KUKA KRL program: MyProgram_282().src

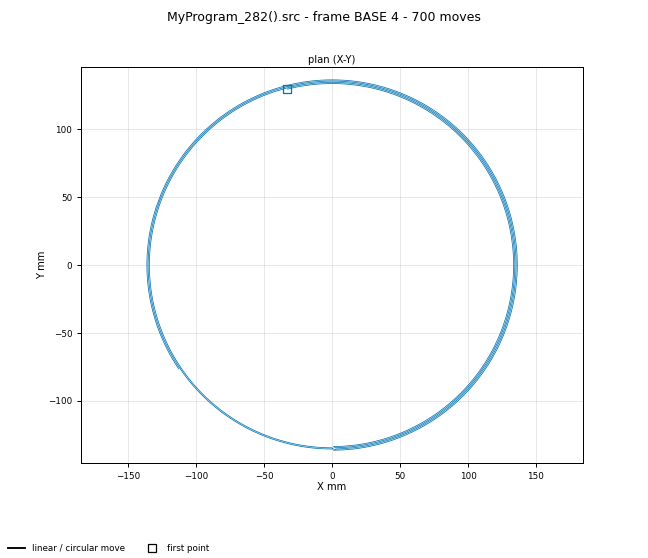
[picture p0: tool path of MyProgram_282().src in frame BASE 4, 700 of 700 moves have a stored position in this frame; points joined in program order, loops and branches not executed]
&ACCESS RVP
&REL 1
&PARAM TEMPLATE = C:\KRC\Roboter\Template\vorgabe
&PARAM EDITMASK = *
DEF MyProgram_282()
; ---- Setting reference (Base) ----
$BASE = BASE_DATA[4]

; --------------------------
; ---- Setting tool (TCP) ----
$TOOL = TOOL_DATA[3]
; --------------------------

$VEL.CP = VEL_APROX_PRINT
Startdeposition()
$VEL.CP = VEL_PRINT
LIN {X -32.8605,Y 129.4603,Z 174,A 104.6033,B 7.9033,C 0.0922,E1 7.8666,E2 347.1729} C_DIS
LIN {X -29.8546,Y 130.1864,Z 174,A 103.1963,B 7.9033,C 0.0926,E1 7.8705,E2 348.5885} C_DIS
LIN {X -26.1954,Y 130.9725,Z 174,A 101.6197,B 7.9033,C 0.0912,E1 7.8748,E2 350.1607} C_DIS
LIN {X -22.189,Y 131.7099,Z 174,A 99.8395,B 7.9033,C 0.0908,E1 7.8797,E2 351.9438} C_DIS
LIN {X -18.2739,Y 132.3113,Z 174,A 98.1779,B 7.9033,C 0.0895,E1 7.8843,E2 353.6} C_DIS
LIN {X -15.2811,Y 132.6899,Z 174,A 96.9189,B 7.9033,C 0.0885,E1 7.8877,E2 354.8542} C_DIS
LIN {X -12.4791,Y 132.9819,Z 174,A 95.5561,B 7.9033,C 0.0906,E1 7.8916,E2 356.2345} C_DIS
LIN {X -8.672,Y 133.2849,Z 174,A 93.9612,B 7.9033,C 0.0896,E1 7.896,E2 357.8234} C_DIS
LIN {X -4.9766,Y 133.4734,Z 174,A 92.4821,B 7.9034,C 0.0876,E1 7.9001,E2 359.289} C_DIS
LIN {X -1.8357,Y 133.5539,Z 174,A 90.9432,B 7.9034,C 0.0906,E1 7.9044,E2 360.8497} C_DIS
LIN {X 2.7143,Y 133.5393,Z 174,A 89.1223,B 7.9034,C 0.0885,E1 7.9095,E2 362.6544} C_DIS
LIN {X 5.81,Y 133.4409,Z 174,A 87.8332,B 7.9034,C 0.088,E1 7.9131,E2 363.9384} C_DIS
LIN {X 8.6689,Y 133.2851,Z 174,A 86.4498,B 7.9034,C 0.0908,E1 7.917,E2 365.3395} C_DIS
LIN {X 12.7986,Y 132.9513,Z 174,A 84.7484,B 7.9034,C 0.09,E1 7.9217,E2 367.0313} C_DIS
LIN {X 17.0686,Y 132.471,Z 174,A 82.9134,B 7.9034,C 0.0904,E1 7.9268,E2 368.8647} C_DIS
LIN {X 20.8861,Y 131.9234,Z 174,A 81.3133,B 7.9034,C 0.0902,E1 7.9312,E2 370.4579} C_DIS
LIN {X 23.9959,Y 131.3934,Z 174,A 79.9828,B 7.9034,C 0.0905,E1 7.9348,E2 371.7853} C_DIS
LIN {X 26.722,Y 130.8653,Z 174,A 78.7856,B 7.9034,C 0.0913,E1 7.9381,E2 372.9829} C_DIS
LIN {X 30.0115,Y 130.1506,Z 174,A 77.2899,B 7.9034,C 0.0931,E1 7.9422,E2 374.4842} C_DIS
LIN {X 35.919,Y 128.6452,Z 174,A 74.2087,B 7.9032,C 0.1029,E1 7.9507,E2 377.6197} C_DIS
LIN {X 40.1681,Y 127.3834,Z 174,A 72.9052,B 7.9033,C 0.0943,E1 7.954,E2 378.8525} C_DIS
LIN {X 44.4232,Y 125.9636,Z 174,A 70.9319,B 7.9033,C 0.0969,E1 7.9592,E2 380.8314} C_DIS
LIN {X 46.9395,Y 125.0457,Z 174,A 69.7782,B 7.9033,C 0.0981,E1 7.9622,E2 381.9855} C_DIS
LIN {X 49.9341,Y 123.8803,Z 174,A 68.3607,B 7.9033,C 0.1002,E1 7.9659,E2 383.4074} C_DIS
LIN {X 53.8065,Y 122.2507,Z 174,A 66.6357,B 7.9033,C 0.1009,E1 7.9703,E2 385.1232} C_DIS
LIN {X 56.4761,Y 121.0388,Z 174,A 65.4067,B 7.9033,C 0.1019,E1 7.9734,E2 386.3488} C_DIS
LIN {X 59.2522,Y 119.7035,Z 174,A 64.0434,B 7.9033,C 0.1043,E1 7.9768,E2 387.7169} C_DIS
LIN {X 62.5045,Y 118.0386,Z 174,A 62.4717,B 7.9032,C 0.1065,E1 7.9807,E2 389.2892} C_DIS
LIN {X 66.3312,Y 115.933,Z 174,A 60.5453,B 7.9032,C 0.11,E1 7.9854,E2 391.222} C_DIS
LIN {X 70.0988,Y 113.6948,Z 174,A 58.7645,B 7.9032,C 0.111,E1 7.9897,E2 392.9911} C_DIS
LIN {X 73.636,Y 111.4363,Z 174,A 56.1409,B 7.9028,C 0.1287,E1 7.996,E2 395.712} C_DIS
LIN {X 78.7721,Y 107.8673,Z 174,A 54.0455,B 7.9029,C 0.1226,E1 8.0006,E2 397.7386} C_DIS
LIN {X 81.3969,Y 105.9004,Z 174,A 53.1152,B 7.903,C 0.1163,E1 8.0026,E2 398.6125} C_DIS
LIN {X 83.7862,Y 104.0199,Z 174,A 51.5738,B 7.903,C 0.123,E1 8.006,E2 400.1825} C_DIS
LIN {X 87.2072,Y 101.1689,Z 174,A 49.5214,B 7.9028,C 0.1291,E1 8.0104,E2 402.2521} C_DIS
LIN {X 90.7533,Y 98.0011,Z 174,A 47.6396,B 7.9028,C 0.1301,E1 8.0142,E2 404.1157} C_DIS
LIN {X 94.316,Y 94.5769,Z 174,A 45.4109,B 7.9028,C 0.1364,E1 8.0187,E2 406.3579} C_DIS
LIN {X 97.4887,Y 91.3036,Z 174,A 43.6195,B 7.9027,C 0.1374,E1 8.0221,E2 408.1304} C_DIS
LIN {X 100.3861,Y 88.108,Z 174,A 41.8763,B 7.9027,C 0.1393,E1 8.0253,E2 409.8615} C_DIS
LIN {X 106.7845,Y 80.2334,Z 174,A 37.8971,B 7.9027,C 0.142,E1 8.0323,E2 413.7978} C_DIS
LIN {X 108.9866,Y 77.2156,Z 174,A 35.9263,B 7.9024,C 0.1527,E1 8.0355,E2 415.8136} C_DIS
LIN {X 111.5979,Y 73.3905,Z 174,A 34.0069,B 7.9024,C 0.1562,E1 8.0385,E2 417.7258} C_DIS
LIN {X 114.0459,Y 69.5264,Z 174,A 32.0466,B 7.9023,C 0.1609,E1 8.0414,E2 419.6868} C_DIS
LIN {X 116.2525,Y 65.7705,Z 174,A 30.1922,B 7.9022,C 0.1653,E1 8.044,E2 421.5405} C_DIS
LIN {X 118.3577,Y 61.8967,Z 174,A 28.4516,B 7.9022,C 0.1672,E1 8.0463,E2 423.264} C_DIS
LIN {X 119.9914,Y 58.6685,Z 174,A 26.8129,B 7.902,C 0.1728,E1 8.0483,E2 424.9141} C_DIS
LIN {X 121.9054,Y 54.5784,Z 174,A 24.9705,B 7.902,C 0.176,E1 8.0504,E2 426.7462} C_DIS
LIN {X 123.4751,Y 50.9311,Z 174,A 23.3908,B 7.9019,C 0.1781,E1 8.0521,E2 428.3122} C_DIS
LIN {X 125.7182,Y 45.1079,Z 174,A 20.7446,B 7.9017,C 0.1847,E1 8.0548,E2 430.9564} C_DIS
LIN {X 126.8147,Y 41.9269,Z 174,A 18.9766,B 7.9015,C 0.195,E1 8.0564,E2 432.7645} C_DIS
LIN {X 127.8659,Y 38.6048,Z 174,A 17.7011,B 7.9015,C 0.1948,E1 8.0574,E2 434.0147} C_DIS
LIN {X 129.0774,Y 34.3337,Z 174,A 15.9304,B 7.9015,C 0.1975,E1 8.0587,E2 435.7705} C_DIS
LIN {X 129.9152,Y 31.0146,Z 174,A 14.4948,B 7.9013,C 0.2009,E1 8.0596,E2 437.2033} C_DIS
LIN {X 130.6576,Y 27.7239,Z 174,A 13.0437,B 7.9013,C 0.2051,E1 8.0605,E2 438.656} C_DIS
LIN {X 131.4588,Y 23.6307,Z 174,A 11.3378,B 7.9012,C 0.2085,E1 8.0614,E2 440.3532} C_DIS
LIN {X 132.0148,Y 20.2961,Z 174,A 9.9295,B 7.9011,C 0.2118,E1 8.062,E2 441.7575} C_DIS
LIN {X 132.5279,Y 16.6348,Z 174,A 8.3933,B 7.901,C 0.2153,E1 8.0626,E2 443.289} C_DIS
LIN {X 132.8256,Y 14.0447,Z 174,A 7.3262,B 7.901,C 0.2175,E1 8.0629,E2 444.3508} C_DIS
LIN {X 133.1108,Y 11.0187,Z 174,A 5.9679,B 7.9008,C 0.2223,E1 8.0632,E2 445.7168} C_DIS
LIN {X 133.38,Y 7.0542,Z 174,A 4.2115,B 7.9006,C 0.2283,E1 8.0635,E2 447.4809} C_DIS
LIN {X 133.5214,Y 3.4601,Z 174,A 2.6915,B 7.9005,C 0.2323,E1 8.0637,E2 448.9995} C_DIS
LIN {X 133.5639,Y -0.9026,Z 174,A 0.8942,B 7.9004,C 0.2362,E1 8.0637,E2 450.7894} C_DIS
LIN {X 133.4787,Y -4.8404,Z 174,A -0.7444,B 7.9003,C 0.2401,E1 8.0635,E2 452.4233} C_DIS
LIN {X 133.2455,Y -9.2583,Z 174,A -2.493,B 7.9002,C 0.2426,E1 8.0633,E2 454.1554} C_DIS
LIN {X 132.9721,Y -12.5819,Z 174,A -3.989,B 7.9,C 0.248,E1 8.0629,E2 455.6608} C_DIS
LIN {X 132.5353,Y -16.5773,Z 174,A -5.793,B 7.8998,C 0.2546,E1 8.0623,E2 457.4761} C_DIS
LIN {X 131.9446,Y -20.7496,Z 174,A -7.4738,B 7.8998,C 0.2572,E1 8.0616,E2 459.1431} C_DIS
LIN {X 131.1931,Y -25.0635,Z 174,A -9.2795,B 7.8996,C 0.2611,E1 8.0607,E2 460.9417} C_DIS
LIN {X 130.4706,Y -28.5898,Z 174,A -11.2579,B 7.8992,C 0.2741,E1 8.0595,E2 462.9744} C_DIS
LIN {X 129.5241,Y -32.609,Z 174,A -13.4588,B 7.8987,C 0.2875,E1 8.058,E2 465.229} C_DIS
LIN {X 127.7535,Y -38.9721,Z 174,A -15.0461,B 7.8993,C 0.2709,E1 8.0569,E2 466.6675} C_DIS
LIN {X 126.3542,Y -43.2965,Z 174,A -17.0965,B 7.899,C 0.2783,E1 8.0551,E2 468.7323} C_DIS
LIN {X 125.4037,Y -45.9802,Z 174,A -18.4062,B 7.8988,C 0.2834,E1 8.0538,E2 470.0541} C_DIS
LIN {X 124.4327,Y -48.5413,Z 174,A -19.6423,B 7.8987,C 0.2878,E1 8.0525,E2 471.2987} C_DIS
LIN {X 122.7297,Y -52.6996,Z 174,A -22.5427,B 7.8978,C 0.312,E1 8.0492,E2 474.3193} C_DIS
LIN {X 119.6529,Y -59.3548,Z 174,A -24.6316,B 7.8982,C 0.2997,E1 8.0468,E2 476.2829} C_DIS
LIN {X 117.5355,Y -63.4486,Z 174,A -27.0607,B 7.8977,C 0.3137,E1 8.0436,E2 478.7694} C_DIS
LIN {X 115.2948,Y -67.4346,Z 174,A -28.5676,B 7.8978,C 0.3098,E1 8.0415,E2 480.2227} C_DIS
LIN {X 113.2822,Y -70.7634,Z 174,A -30.2002,B 7.8978,C 0.3133,E1 8.0391,E2 481.8526} C_DIS
LIN {X 111.0915,Y -74.1547,Z 174,A -32.0728,B 7.8974,C 0.3203,E1 8.0362,E2 483.7441} C_DIS
LIN {X 108.8221,Y -77.4473,Z 174,A -33.5927,B 7.8974,C 0.3207,E1 8.0338,E2 485.2418} C_DIS
LIN {X 105.9642,Y -81.3135,Z 174,A -35.6174,B 7.8973,C 0.3248,E1 8.0304,E2 487.2639} C_DIS
LIN {X 103.3829,Y -84.5709,Z 174,A -37.7765,B 7.8968,C 0.3362,E1 8.0266,E2 489.4709} C_DIS
LIN {X 100.559,Y -87.9099,Z 174,A -39.1592,B 7.897,C 0.3309,E1 8.0241,E2 490.7949} C_DIS
LIN {X 97.7749,Y -90.9962,Z 174,A -40.9704,B 7.8968,C 0.3354,E1 8.0207,E2 492.6113} C_DIS
LIN {X 94.5935,Y -94.2993,Z 174,A -43.2946,B 7.8963,C 0.3464,E1 8.0161,E2 494.9812} C_DIS
LIN {X 91.5907,Y -97.218,Z 174,A -44.4878,B 7.8967,C 0.3386,E1 8.0138,E2 496.1019} C_DIS
LIN {X 89.06,Y -99.5418,Z 174,A -46.1353,B 7.8964,C 0.3449,E1 8.0103,E2 497.7723} C_DIS
LIN {X 85.8583,Y -102.3162,Z 174,A -47.9147,B 7.8963,C 0.3477,E1 8.0066,E2 499.5487} C_DIS
LIN {X 80.6674,Y -106.457,Z 174,A -50.7613,B 7.896,C 0.353,E1 8.0003,E2 502.3976} C_DIS
LIN {X 76.336,Y -109.6042,Z 174,A -53.0261,B 7.8959,C 0.3564,E1 7.9952,E2 504.6606} C_DIS
LIN {X 72.5931,Y -112.1183,Z 174,A -54.9381,B 7.8958,C 0.3593,E1 7.9907,E2 506.5715} C_DIS
LIN {X 67.02,Y -115.5361,Z 174,A -58.2995,B 7.8951,C 0.374,E1 7.9825,E2 510.0037} C_DIS
LIN {X 62.4489,Y -118.0678,Z 174,A -59.6683,B 7.8957,C 0.3612,E1 7.9794,E2 511.2669} C_DIS
LIN {X 58.5733,Y -120.0384,Z 174,A -61.6545,B 7.8955,C 0.3661,E1 7.9744,E2 513.2697} C_DIS
LIN {X 55.9982,Y -121.2598,Z 174,A -62.9844,B 7.8953,C 0.3696,E1 7.971,E2 514.6139} C_DIS
LIN {X 52.5607,Y -122.7898,Z 174,A -64.4615,B 7.8953,C 0.3692,E1 7.9672,E2 516.0753} C_DIS
LIN {X 49.6424,Y -123.9978,Z 174,A -65.8929,B 7.8952,C 0.3722,E1 7.9635,E2 517.5172} C_DIS
LIN {X 46.351,Y -125.2662,Z 174,A -67.3152,B 7.8952,C 0.3722,E1 7.9598,E2 518.9295} C_DIS
LIN {X 42.9664,Y -126.4684,Z 174,A -68.8545,B 7.8951,C 0.3739,E1 7.9558,E2 520.4698} C_DIS
LIN {X 40.2953,Y -127.3428,Z 174,A -70.1004,B 7.8951,C 0.3758,E1 7.9524,E2 521.7215} C_DIS
LIN {X 36.0701,Y -128.603,Z 174,A -72.0478,B 7.8949,C 0.3785,E1 7.9472,E2 523.6771} C_DIS
LIN {X 32.3796,Y -129.5823,Z 174,A -73.5717,B 7.8949,C 0.3779,E1 7.9431,E2 525.1881} C_DIS
LIN {X 29.4655,Y -130.2753,Z 174,A -74.7848,B 7.8949,C 0.3776,E1 7.9398,E2 526.393} C_DIS
LIN {X 26.6085,Y -130.8884,Z 174,A -76.0796,B 7.8949,C 0.3792,E1 7.9363,E2 527.6938} C_DIS
LIN {X 23.365,Y -131.5063,Z 174,A -77.5523,B 7.8947,C 0.3811,E1 7.9322,E2 529.1744} C_DIS
LIN {X 19.6691,Y -132.1119,Z 174,A -79.2862,B 7.8946,C 0.3842,E1 7.9274,E2 530.9251} C_DIS
LIN {X 16.1177,Y -132.5901,Z 174,A -80.7356,B 7.8946,C 0.3835,E1 7.9234,E2 532.3645} C_DIS
LIN {X 11.8861,Y -133.0375,Z 174,A -82.3975,B 7.8947,C 0.3814,E1 7.9188,E2 534.0072} C_DIS
LIN {X 9.1903,Y -133.2504,Z 174,A -83.8262,B 7.8945,C 0.3864,E1 7.9147,E2 535.4697} C_DIS
LIN {X 5.1786,Y -133.4655,Z 174,A -85.4054,B 7.8945,C 0.3843,E1 7.9104,E2 537.032} C_DIS
LIN {X 0.9674,Y -133.5612,Z 174,A -86.8361,B 7.8949,C 0.3782,E1 7.9065,E2 538.4169} C_DIS
Enddeposition()
LIN {X 0.9674,Y -133.5612,Z 174,A -86.8361,B 7.8949,C 0.3782,E1 7.9065,E2 538.4169} C_DIS
Startdeposition()
$VEL.CP = VEL_PRINT
LIN {X 2.3813,Y -134.4521,Z 174,A -85.842,B 7.8949,C 0.3759,E1 7.9092,E2 537.4069} C_DIS
LIN {X 8.4172,Y -134.2094,Z 174,A -83.691,B 7.8946,C 0.3827,E1 7.9151,E2 535.3077} C_DIS
LIN {X 14.1408,Y -133.7276,Z 174,A -80.8337,B 7.8949,C 0.3746,E1 7.9232,E2 532.3976} C_DIS
LIN {X 17.6758,Y -133.3063,Z 174,A -79.3415,B 7.8949,C 0.3743,E1 7.9273,E2 530.9077} C_DIS
LIN {X 21.007,Y -132.8226,Z 174,A -77.9448,B 7.8949,C 0.3741,E1 7.9311,E2 529.5149} C_DIS
LIN {X 23.717,Y -132.3649,Z 174,A -76.7694,B 7.895,C 0.3733,E1 7.9344,E2 528.3381} C_DIS
LIN {X 26.9602,Y -131.7426,Z 174,A -75.349,B 7.895,C 0.3721,E1 7.9383,E2 526.9152} C_DIS
LIN {X 30.122,Y -131.0558,Z 174,A -74.0054,B 7.895,C 0.3717,E1 7.9419,E2 525.5751} C_DIS
LIN {X 33.8293,Y -130.1503,Z 174,A -72.2161,B 7.8953,C 0.3674,E1 7.9468,E2 523.7641} C_DIS
LIN {X 37.6768,Y -129.0867,Z 174,A -70.661,B 7.8953,C 0.3686,E1 7.951,E2 522.2262} C_DIS
LIN {X 41.2611,Y -127.9865,Z 174,A -69.0904,B 7.8953,C 0.3675,E1 7.9551,E2 520.6579} C_DIS
LIN {X 44.3458,Y -126.9506,Z 174,A -67.7307,B 7.8953,C 0.3665,E1 7.9587,E2 519.3005} C_DIS
LIN {X 47.4826,Y -125.8109,Z 174,A -66.3275,B 7.8953,C 0.3653,E1 7.9624,E2 517.8986} C_DIS
LIN {X 50.4496,Y -124.6505,Z 174,A -64.9177,B 7.8955,C 0.3627,E1 7.9661,E2 516.4812} C_DIS
LIN {X 53.3913,Y -123.4189,Z 174,A -63.5797,B 7.8955,C 0.3614,E1 7.9695,E2 515.1447} C_DIS
LIN {X 57.2513,Y -121.679,Z 174,A -61.6065,B 7.8958,C 0.3559,E1 7.9746,E2 513.1488} C_DIS
LIN {X 60.8457,Y -119.9195,Z 174,A -60.1362,B 7.8958,C 0.3579,E1 7.9782,E2 511.7067} C_DIS
LIN {X 64.7447,Y -117.8619,Z 174,A -57.9241,B 7.8961,C 0.3488,E1 7.9837,E2 509.4509} C_DIS
LIN {X 67.8779,Y -116.0865,Z 174,A -56.5245,B 7.8961,C 0.349,E1 7.9871,E2 508.0671} C_DIS
LIN {X 71.2194,Y -114.0668,Z 174,A -55.0969,B 7.8961,C 0.3508,E1 7.9904,E2 506.6679} C_DIS
LIN {X 74.4195,Y -112.0055,Z 174,A -53.4031,B 7.8962,C 0.3468,E1 7.9944,E2 504.9635} C_DIS
LIN {X 78.1874,Y -109.4081,Z 174,A -51.4969,B 7.8963,C 0.3442,E1 7.9987,E2 503.0612} C_DIS
LIN {X 82.2337,Y -106.4004,Z 174,A -49.2415,B 7.8966,C 0.3382,E1 8.0038,E2 500.7903} C_DIS
LIN {X 85.1332,Y -104.0948,Z 174,A -47.7998,B 7.8966,C 0.3378,E1 8.0069,E2 499.3644} C_DIS
LIN {X 88.4233,Y -101.3149,Z 174,A -45.9787,B 7.8967,C 0.3345,E1 8.0107,E2 497.5434} C_DIS
LIN {X 91.8873,Y -98.1847,Z 174,A -43.8328,B 7.897,C 0.3274,E1 8.0152,E2 495.3758} C_DIS
LIN {X 95.0883,Y -95.0883,Z 174,A -42.2035,B 7.897,C 0.3287,E1 8.0183,E2 493.7786} C_DIS
LIN {X 97.9798,Y -92.1054,Z 174,A -40.4175,B 7.8972,C 0.3245,E1 8.0218,E2 491.9888} C_DIS
LIN {X 100.9496,Y -88.8407,Z 174,A -38.3676,B 7.8975,C 0.317,E1 8.0256,E2 489.9158} C_DIS
LIN {X 103.8494,Y -85.4336,Z 174,A -36.7918,B 7.8974,C 0.3192,E1 8.0284,E2 488.3798} C_DIS
LIN {X 106.1126,Y -82.6051,Z 174,A -34.9879,B 7.8977,C 0.3104,E1 8.0316,E2 486.5415} C_DIS
LIN {X 108.9982,Y -78.758,Z 174,A -32.7842,B 7.898,C 0.3025,E1 8.0352,E2 484.3163} C_DIS
LIN {X 111.3244,Y -75.4339,Z 174,A -31.7902,B 7.8976,C 0.3129,E1 8.0367,E2 483.413} C_DIS
LIN {X 112.9455,Y -72.9849,Z 174,A -30.1105,B 7.8981,C 0.3013,E1 8.0393,E2 481.6784} C_DIS
LIN {X 114.9785,Y -69.738,Z 174,A -28.6361,B 7.8981,C 0.3003,E1 8.0414,E2 480.2222} C_DIS
LIN {X 118.6158,Y -63.3546,Z 174,A -25.506,B 7.8984,C 0.2923,E1 8.0457,E2 477.0891} C_DIS
LIN {X 121.6414,Y -57.3288,Z 174,A -22.2905,B 7.8989,C 0.2779,E1 8.0497,E2 473.8275} C_DIS
LIN {X 123.3919,Y -53.4539,Z 174,A -21.2791,B 7.8985,C 0.2891,E1 8.0507,E2 472.9147} C_DIS
LIN {X 124.8493,Y -49.9564,Z 174,A -19.4436,B 7.8988,C 0.2803,E1 8.0527,E2 471.0501} C_DIS
LIN {X 125.9847,Y -47.0186,Z 174,A -18.1067,B 7.899,C 0.2767,E1 8.054,E2 469.7125} C_DIS
LIN {X 127.049,Y -44.0619,Z 174,A -16.7581,B 7.899,C 0.2729,E1 8.0553,E2 468.3614} C_DIS
LIN {X 128.2227,Y -40.5219,Z 174,A -15.1119,B 7.8993,C 0.2673,E1 8.0567,E2 466.7065} C_DIS
LIN {X 130.3883,Y -32.8914,Z 174,A -11.9004,B 7.8995,C 0.2612,E1 8.0591,E2 463.5128} C_DIS
LIN {X 131.0796,Y -30.0178,Z 174,A -10.6649,B 7.8995,C 0.2582,E1 8.0598,E2 462.2791} C_DIS
LIN {X 131.7739,Y -26.8062,Z 174,A -9.2631,B 7.8997,C 0.2541,E1 8.0606,E2 460.8758} C_DIS
LIN {X 132.4425,Y -23.2829,Z 174,A -7.6806,B 7.8999,C 0.2487,E1 8.0614,E2 459.285} C_DIS
LIN {X 133.1232,Y -19.0049,Z 174,A -5.9996,B 7.8999,C 0.2467,E1 8.0621,E2 457.6228} C_DIS
LIN {X 133.5736,Y -15.5317,Z 174,A -4.5641,B 7.9,C 0.2436,E1 8.0626,E2 456.193} C_DIS
LIN {X 133.9202,Y -12.1981,Z 174,A -3.135,B 7.9002,C 0.2394,E1 8.063,E2 454.7624} C_DIS
LIN {X 134.3453,Y -5.8976,Z 174,A -0.5351,B 7.9003,C 0.2335,E1 8.0635,E2 452.1714} C_DIS
LIN {X 134.4584,Y -2.0056,Z 174,A 1.1198,B 7.9005,C 0.2288,E1 8.0635,E2 450.5155} C_DIS
LIN {X 134.4696,Y 1.1061,Z 174,A 2.4735,B 7.9006,C 0.2244,E1 8.0635,E2 449.1573} C_DIS
LIN {X 134.3394,Y 6.036,Z 174,A 4.4801,B 7.9007,C 0.2203,E1 8.0634,E2 447.1606} C_DIS
LIN {X 134.071,Y 10.4088,Z 174,A 6.3941,B 7.9009,C 0.2139,E1 8.063,E2 445.2392} C_DIS
LIN {X 133.7055,Y 14.3466,Z 174,A 8.0408,B 7.901,C 0.2099,E1 8.0626,E2 443.5958} C_DIS
LIN {X 133.2842,Y 17.8447,Z 174,A 9.5869,B 7.9011,C 0.2047,E1 8.062,E2 442.0429} C_DIS
LIN {X 132.6696,Y 21.9493,Z 174,A 11.238,B 7.9012,C 0.202,E1 8.0613,E2 440.4049} C_DIS
LIN {X 132.0391,Y 25.4689,Z 174,A 12.7066,B 7.9012,C 0.1988,E1 8.0605,E2 438.9419} C_DIS
LIN {X 131.3327,Y 28.8953,Z 174,A 14.17,B 7.9014,C 0.1952,E1 8.0597,E2 437.4807} C_DIS
LIN {X 130.4583,Y 32.6158,Z 174,A 15.8511,B 7.9015,C 0.1896,E1 8.0586,E2 435.7919} C_DIS
LIN {X 129.4257,Y 36.4964,Z 174,A 17.4995,B 7.9015,C 0.1861,E1 8.0574,E2 434.15} C_DIS
LIN {X 128.0732,Y 40.9899,Z 174,A 19.4535,B 7.9017,C 0.1815,E1 8.0558,E2 432.2002} C_DIS
LIN {X 126.8433,Y 44.6551,Z 174,A 21.7743,B 7.9021,C 0.1636,E1 8.0536,E2 429.7949} C_DIS
LIN {X 124.8933,Y 49.8474,Z 174,A 23.2295,B 7.9018,C 0.1753,E1 8.0522,E2 428.4506} C_DIS
LIN {X 123.3919,Y 53.4539,Z 174,A 25.0313,B 7.902,C 0.1682,E1 8.0502,E2 426.6308} C_DIS
LIN {X 121.9697,Y 56.6241,Z 174,A 26.4792,B 7.902,C 0.165,E1 8.0485,E2 425.186} C_DIS
LIN {X 120.3103,Y 60.0725,Z 174,A 28.033,B 7.9021,C 0.1623,E1 8.0466,E2 423.6407} C_DIS
LIN {X 119.1138,Y 62.4081,Z 174,A 29.1522,B 7.9021,C 0.1594,E1 8.0452,E2 422.5207} C_DIS
LIN {X 117.0655,Y 66.1754,Z 174,A 31.0938,B 7.9023,C 0.1526,E1 8.0425,E2 420.5641} C_DIS
LIN {X 114.7688,Y 70.0828,Z 174,A 32.9901,B 7.9023,C 0.1486,E1 8.0398,E2 418.6711} C_DIS
LIN {X 112.2911,Y 73.9872,Z 174,A 34.8991,B 7.9025,C 0.145,E1 8.0369,E2 416.7687} C_DIS
LIN {X 109.719,Y 77.7506,Z 174,A 36.7459,B 7.9025,C 0.1423,E1 8.034,E2 414.9326} C_DIS
LIN {X 107.2283,Y 81.1512,Z 174,A 38.9497,B 7.9027,C 0.1303,E1 8.0302,E2 412.678} C_DIS
LIN {X 104.6851,Y 84.4061,Z 174,A 40.4134,B 7.9027,C 0.1321,E1 8.0277,E2 411.2501} C_DIS
LIN {X 102.145,Y 87.4639,Z 174,A 42.0062,B 7.9027,C 0.1303,E1 8.0249,E2 409.669} C_DIS
LIN {X 99.1956,Y 90.7949,Z 174,A 43.8858,B 7.9027,C 0.1266,E1 8.0214,E2 407.7907} C_DIS
LIN {X 95.8545,Y 94.3152,Z 174,A 45.6568,B 7.9027,C 0.128,E1 8.018,E2 406.0553} C_DIS
LIN {X 92.6153,Y 97.4985,Z 174,A 47.8455,B 7.9029,C 0.1193,E1 8.0136,E2 403.8352} C_DIS
LIN {X 89.0835,Y 100.735,Z 174,A 49.7474,B 7.9029,C 0.118,E1 8.0096,E2 401.9497} C_DIS
LIN {X 86.0762,Y 103.3172,Z 174,A 51.4874,B 7.9029,C 0.114,E1 8.0059,E2 400.2031} C_DIS
LIN {X 82.7455,Y 106.0035,Z 174,A 53.3315,B 7.903,C 0.1103,E1 8.0019,E2 398.3562} C_DIS
LIN {X 80.0111,Y 108.0822,Z 174,A 54.7695,B 7.903,C 0.1083,E1 7.9987,E2 396.921} C_DIS
LIN {X 75.6484,Y 111.1792,Z 174,A 57.0117,B 7.903,C 0.1053,E1 7.9935,E2 394.6831} C_DIS
LIN {X 71.9678,Y 113.5962,Z 174,A 58.8795,B 7.9031,C 0.1025,E1 7.9891,E2 392.8161} C_DIS
LIN {X 68.0663,Y 115.9758,Z 174,A 60.7919,B 7.9031,C 0.1003,E1 7.9846,E2 390.9079} C_DIS
LIN {X 64.0541,Y 118.2397,Z 174,A 62.7306,B 7.9031,C 0.098,E1 7.9798,E2 388.9721} C_DIS
LIN {X 60.8995,Y 119.8921,Z 174,A 64.1407,B 7.9031,C 0.098,E1 7.9764,E2 387.5749} C_DIS
LIN {X 58.0887,Y 121.279,Z 174,A 65.5291,B 7.9032,C 0.0953,E1 7.9729,E2 386.1801} C_DIS
LIN {X 54.8131,Y 122.7941,Z 174,A 67.0554,B 7.9032,C 0.0937,E1 7.969,E2 384.6552} C_DIS
LIN {X 51.3445,Y 124.2855,Z 174,A 68.7308,B 7.9032,C 0.0908,E1 7.9647,E2 382.9719} C_DIS
LIN {X 47.7987,Y 125.6926,Z 174,A 70.2135,B 7.9032,C 0.0916,E1 7.9608,E2 381.5067} C_DIS
LIN {X 43.8151,Y 127.1345,Z 174,A 72.0448,B 7.9032,C 0.0894,E1 7.956,E2 379.6725} C_DIS
LIN {X 37.4065,Y 129.1659,Z 174,A 74.869,B 7.9032,C 0.0878,E1 7.9485,E2 376.8537} C_DIS
LIN {X 34.4529,Y 129.9844,Z 174,A 76.1582,B 7.9032,C 0.0871,E1 7.945,E2 375.5668} C_DIS
LIN {X 31.121,Y 130.8227,Z 174,A 77.5904,B 7.9033,C 0.0866,E1 7.9411,E2 374.1388} C_DIS
LIN {X 27.4201,Y 131.649,Z 174,A 79.3043,B 7.9033,C 0.084,E1 7.9364,E2 372.4135} C_DIS
LIN {X 23.7136,Y 132.3655,Z 174,A 80.8085,B 7.9033,C 0.0849,E1 7.9323,E2 370.9223} C_DIS
LIN {X 19.8449,Y 133.0026,Z 174,A 82.625,B 7.9033,C 0.0817,E1 7.9273,E2 369.0888} C_DIS
LIN {X 16.0053,Y 133.5171,Z 174,A 84.1357,B 7.9033,C 0.0835,E1 7.9231,E2 367.5954} C_DIS
LIN {X 12.5603,Y 133.8854,Z 174,A 85.601,B 7.9033,C 0.0832,E1 7.9191,E2 366.1319} C_DIS
LIN {X 8.953,Y 134.1764,Z 174,A 87.2671,B 7.9033,C 0.0809,E1 7.9144,E2 364.4515} C_DIS
LIN {X 4.969,Y 134.3815,Z 174,A 88.8768,B 7.9033,C 0.0822,E1 7.9099,E2 362.8534} C_DIS
LIN {X -0.5309,Y 134.4723,Z 174,A 91.219,B 7.9033,C 0.0822,E1 7.9034,E2 360.5125} C_DIS
LIN {X -4.0382,Y 134.4128,Z 174,A 92.8113,B 7.9033,C 0.0806,E1 7.8989,E2 358.9091} C_DIS
LIN {X -8.3743,Y 134.2121,Z 174,A 94.5206,B 7.9033,C 0.0832,E1 7.8942,E2 357.2175} C_DIS
LIN {X -12.2442,Y 133.9158,Z 174,A 96.3017,B 7.9033,C 0.0816,E1 7.8892,E2 355.4221} C_DIS
LIN {X -16.1828,Y 133.4959,Z 174,A 97.8683,B 7.9033,C 0.0841,E1 7.8849,E2 353.8708} C_DIS
LIN {X -19.1868,Y 133.0972,Z 174,A 99.1997,B 7.9033,C 0.084,E1 7.8812,E2 352.5354} C_DIS
LIN {X -22.3361,Y 132.605,Z 174,A 100.5591,B 7.9033,C 0.0846,E1 7.8775,E2 351.1766} C_DIS
LIN {X -26.3997,Y 131.8566,Z 174,A 102.3847,B 7.9033,C 0.0846,E1 7.8724,E2 349.3442} C_DIS
LIN {X -30.1179,Y 131.0567,Z 174,A 103.9525,B 7.9033,C 0.0864,E1 7.8682,E2 347.7837} C_DIS
LIN {X -33.4639,Y 130.243,Z 174,A 105.4104,B 7.9033,C 0.0876,E1 7.8642,E2 346.328} C_DIS
LIN {X -42.2849,Y 127.6516,Z 174,A 110.6048,B 7.9035,C 0.0708,E1 7.85,E2 340.9811} C_DIS
LIN {X -50.053,Y 124.8104,Z 174,A 112.9823,B 7.9032,C 0.0925,E1 7.8442,E2 338.746} C_DIS
LIN {X -53.7812,Y 123.2504,Z 174,A 114.6321,B 7.9032,C 0.0955,E1 7.84,E2 337.1061} C_DIS
LIN {X -57.5211,Y 121.5501,Z 174,A 117.135,B 7.9033,C 0.0862,E1 7.8334,E2 334.5136} C_DIS
LIN {X -62.4517,Y 119.0909,Z 174,A 118.7522,B 7.9031,C 0.1004,E1 7.8296,E2 332.9867} C_DIS
LIN {X -66.276,Y 117.0088,Z 174,A 120.6779,B 7.9031,C 0.102,E1 7.8249,E2 331.0542} C_DIS
LIN {X -69.7149,Y 114.9924,Z 174,A 122.5742,B 7.9031,C 0.1016,E1 7.8203,E2 329.1354} C_DIS
LIN {X -73.5924,Y 112.551,Z 174,A 124.4486,B 7.9031,C 0.1058,E1 7.8159,E2 327.2721} C_DIS
LIN {X -78.2444,Y 109.3674,Z 174,A 126.8243,B 7.9031,C 0.1102,E1 7.8105,E2 324.9016} C_DIS
LIN {X -81.2312,Y 107.1679,Z 174,A 128.3699,B 7.903,C 0.1134,E1 7.8071,E2 323.3616} C_DIS
LIN {X -84.4073,Y 104.6843,Z 174,A 130.0713,B 7.903,C 0.1168,E1 7.8033,E2 321.6637} C_DIS
LIN {X -87.4332,Y 102.1715,Z 174,A 132.1851,B 7.903,C 0.1135,E1 7.7987,E2 319.4986} C_DIS
LIN {X -90.2359,Y 99.7041,Z 174,A 133.3286,B 7.9028,C 0.1231,E1 7.7965,E2 318.4106} C_DIS
LIN {X -92.9859,Y 97.1443,Z 174,A 135.2172,B 7.9028,C 0.1222,E1 7.7926,E2 316.4888} C_DIS
LIN {X -95.8367,Y 94.3334,Z 174,A 136.8478,B 7.9028,C 0.1268,E1 7.7894,E2 314.8689} C_DIS
LIN {X -99.5704,Y 90.3833,Z 174,A 139.006,B 7.9026,C 0.134,E1 7.7853,E2 312.7319} C_DIS
LIN {X -102.0372,Y 87.5891,Z 174,A 140.8975,B 7.9026,C 0.1331,E1 7.7818,E2 310.8054} C_DIS
LIN {X -104.3536,Y 84.8166,Z 174,A 142.3734,B 7.9026,C 0.1375,E1 7.7792,E2 309.3386} C_DIS
LIN {X -107.1068,Y 81.3123,Z 174,A 144.2931,B 7.9026,C 0.1415,E1 7.7759,E2 307.4182} C_DIS
LIN {X -109.554,Y 77.9834,Z 174,A 146.0587,B 7.9024,C 0.1456,E1 7.773,E2 305.6536} C_DIS
LIN {X -112.0702,Y 74.3225,Z 174,A 147.9557,B 7.9024,C 0.1501,E1 7.7701,E2 303.758} C_DIS
LIN {X -114.6831,Y 70.2222,Z 174,A 150.219,B 7.9024,C 0.1525,E1 7.7667,E2 301.4735} C_DIS
LIN {X -116.9969,Y 66.2967,Z 174,A 152.4472,B 7.9023,C 0.1534,E1 7.7635,E2 299.2123} C_DIS
LIN {X -118.8895,Y 62.8353,Z 174,A 153.5059,B 7.902,C 0.1664,E1 7.7623,E2 298.2308} C_DIS
LIN {X -120.648,Y 59.388,Z 174,A 155.3959,B 7.902,C 0.1673,E1 7.7598,E2 296.3132} C_DIS
LIN {X -122.1317,Y 56.2738,Z 174,A 156.8719,B 7.902,C 0.1711,E1 7.7581,E2 294.838} C_DIS
LIN {X -123.5734,Y 53.0341,Z 174,A 158.4305,B 7.9019,C 0.1744,E1 7.7563,E2 293.275} C_DIS
LIN {X -125.2331,Y 48.986,Z 174,A 160.9132,B 7.9019,C 0.1709,E1 7.7537,E2 290.7188} C_DIS
LIN {X -126.9254,Y 44.4184,Z 174,A 162.2385,B 7.9016,C 0.1869,E1 7.7526,E2 289.4869} C_DIS
LIN {X -128.222,Y 40.524,Z 174,A 164.1958,B 7.9016,C 0.1889,E1 7.7508,E2 287.5061} C_DIS
LIN {X -129.2305,Y 37.1856,Z 174,A 165.6964,B 7.9014,C 0.1928,E1 7.7497,E2 286.0052} C_DIS
LIN {X -130.0577,Y 34.1782,Z 174,A 167.0568,B 7.9014,C 0.1961,E1 7.7487,E2 284.6422} C_DIS
LIN {X -130.7645,Y 31.3625,Z 174,A 168.327,B 7.9013,C 0.1991,E1 7.7478,E2 283.3691} C_DIS
LIN {X -131.657,Y 27.3807,Z 174,A 170.175,B 7.9012,C 0.2025,E1 7.7467,E2 281.5095} C_DIS
LIN {X -132.349,Y 23.8058,Z 174,A 171.6825,B 7.9011,C 0.2075,E1 7.746,E2 280.0088} C_DIS
LIN {X -132.9284,Y 20.3242,Z 174,A 173.2849,B 7.901,C 0.2105,E1 7.7453,E2 278.3958} C_DIS
LIN {X -133.5099,Y 16.0657,Z 174,A 175.0881,B 7.9008,C 0.2161,E1 7.7446,E2 276.5977} C_DIS
LIN {X -133.9018,Y 12.3901,Z 174,A 176.7815,B 7.9008,C 0.219,E1 7.7441,E2 274.8913} C_DIS
LIN {X -134.2173,Y 8.2887,Z 174,A 178.471,B 7.9006,C 0.2249,E1 7.7438,E2 273.2111} C_DIS
LIN {X -134.395,Y 4.6238,Z 174,A -179.8037,B 7.9006,C 0.2272,E1 7.7436,E2 271.4675} C_DIS
LIN {X -134.4765,Y 0.1063,Z 174,A -177.8878,B 7.9004,C 0.2329,E1 7.7436,E2 269.5544} C_DIS
LIN {X -134.4198,Y -3.7854,Z 174,A -176.297,B 7.9002,C 0.2386,E1 7.7436,E2 267.9732} C_DIS
LIN {X -134.2674,Y -7.4689,Z 174,A -174.5566,B 7.9002,C 0.2408,E1 7.7439,E2 266.2134} C_DIS
LIN {X -133.9841,Y -11.4568,Z 174,A -172.9515,B 7.8999,C 0.247,E1 7.7443,E2 264.6217} C_DIS
LIN {X -133.6903,Y -14.4878,Z 174,A -171.5928,B 7.8999,C 0.2499,E1 7.7447,E2 263.2567} C_DIS
LIN {X -133.1721,Y -18.6626,Z 174,A -169.7202,B 7.8997,C 0.2539,E1 7.7454,E2 261.3757} C_DIS
LIN {X -132.5898,Y -22.4271,Z 174,A -168.1743,B 7.8995,C 0.2596,E1 7.746,E2 259.8406} C_DIS
LIN {X -131.9805,Y -25.7756,Z 174,A -166.6562,B 7.8995,C 0.2627,E1 7.7468,E2 258.3152} C_DIS
LIN {X -131.187,Y -29.5476,Z 174,A -164.3928,B 7.8995,C 0.2587,E1 7.7483,E2 255.9763} C_DIS
LIN {X -130.0374,Y -34.2544,Z 174,A -162.859,B 7.8991,C 0.2718,E1 7.7493,E2 254.5097} C_DIS
LIN {X -128.241,Y -40.4645,Z 174,A -160.238,B 7.8988,C 0.2812,E1 7.7514,E2 251.9072} C_DIS
LIN {X -126.9395,Y -44.3777,Z 174,A -158.1978,B 7.8988,C 0.282,E1 7.7532,E2 249.8333} C_DIS
LIN {X -125.7762,Y -47.5753,Z 174,A -156.8476,B 7.8986,C 0.2873,E1 7.7545,E2 248.4964} C_DIS
LIN {X -124.6749,Y -50.389,Z 174,A -155.5745,B 7.8985,C 0.2909,E1 7.7558,E2 247.2258} C_DIS
LIN {X -123.3315,Y -53.5935,Z 174,A -153.9703,B 7.8984,C 0.293,E1 7.7576,E2 245.6073} C_DIS
LIN {X -120.6633,Y -59.357,Z 174,A -151.4685,B 7.898,C 0.3029,E1 7.7605,E2 243.1324} C_DIS
LIN {X -118.9991,Y -62.6265,Z 174,A -148.8803,B 7.8984,C 0.2921,E1 7.7641,E2 240.4177} C_DIS
LIN {X -116.1285,Y -67.8064,Z 174,A -147.2994,B 7.8977,C 0.312,E1 7.7661,E2 238.9556} C_DIS
LIN {X -113.7521,Y -71.7208,Z 174,A -145.0274,B 7.8977,C 0.312,E1 7.7695,E2 236.6449} C_DIS
LIN {X -110.1713,Y -77.1091,Z 174,A -142.2408,B 7.8974,C 0.318,E1 7.7738,E2 233.8559} C_DIS
LIN {X -107.8152,Y -80.3696,Z 174,A -140.1711,B 7.8974,C 0.3167,E1 7.7773,E2 231.7426} C_DIS
LIN {X -105.4426,Y -83.459,Z 174,A -139.0476,B 7.897,C 0.3283,E1 7.7792,E2 230.6866} C_DIS
LIN {X -103.3592,Y -86.0255,Z 174,A -137.3616,B 7.897,C 0.3272,E1 7.7822,E2 228.9666} C_DIS
LIN {X -100.1573,Y -89.7325,Z 174,A -135.4835,B 7.8967,C 0.3347,E1 7.7856,E2 227.1153} C_DIS
LIN {X -97.3539,Y -92.7667,Z 174,A -133.7883,B 7.8965,C 0.3393,E1 7.7888,E2 225.4288} C_DIS
LIN {X -95.1856,Y -94.9904,Z 174,A -132.1045,B 7.8967,C 0.3365,E1 7.7922,E2 223.7005} C_DIS
LIN {X -91.9977,Y -98.0813,Z 174,A -130.2462,B 7.8965,C 0.3406,E1 7.7959,E2 221.8469} C_DIS
LIN {X -89.0056,Y -100.8038,Z 174,A -128.5053,B 7.8964,C 0.3435,E1 7.7996,E2 220.1042} C_DIS
LIN {X -85.6437,Y -103.6753,Z 174,A -126.0884,B 7.8966,C 0.3387,E1 7.8049,E2 217.6209} C_DIS
LIN {X -81.9363,Y -106.6299,Z 174,A -123.8236,B 7.8966,C 0.3383,E1 7.81,E2 215.3256} C_DIS
LIN {X -77.1785,Y -110.1229,Z 174,A -122.0345,B 7.8959,C 0.3535,E1 7.8139,E2 213.6281} C_DIS
LIN {X -73.6159,Y -112.5356,Z 174,A -120.1102,B 7.8959,C 0.3549,E1 7.8184,E2 211.6927} C_DIS
LIN {X -69.8751,Y -114.8955,Z 174,A -118.2017,B 7.8957,C 0.3572,E1 7.8229,E2 209.7812} C_DIS
LIN {X -65.979,Y -117.1759,Z 174,A -116.3039,B 7.8957,C 0.3602,E1 7.8275,E2 207.8867} C_DIS
LIN {X -62.2518,Y -119.1958,Z 174,A -114.572,B 7.8955,C 0.3636,E1 7.8317,E2 206.164} C_DIS
LIN {X -58.9149,Y -120.8813,Z 174,A -112.9803,B 7.8954,C 0.3655,E1 7.8357,E2 204.5725} C_DIS
LIN {X -56.1724,Y -122.1786,Z 174,A -111.6484,B 7.8954,C 0.3663,E1 7.8391,E2 203.2356} C_DIS
LIN {X -52.2686,Y -123.8996,Z 174,A -109.972,B 7.8951,C 0.3705,E1 7.8434,E2 201.5768} C_DIS
LIN {X -49.1087,Y -125.1854,Z 174,A -108.2002,B 7.8953,C 0.3667,E1 7.8481,E2 199.7649} C_DIS
LIN {X -44.7873,Y -126.7975,Z 174,A -105.8339,B 7.8955,C 0.3619,E1 7.8544,E2 197.3477} C_DIS
LIN {X -40.4688,Y -128.2396,Z 174,A -104.3872,B 7.8951,C 0.3715,E1 7.8581,E2 195.963} C_DIS
LIN {X -37.4138,Y -129.1637,Z 174,A -103.1151,B 7.895,C 0.3739,E1 7.8615,E2 194.7016} C_DIS
LIN {X -34.4249,Y -129.9919,Z 174,A -101.7714,B 7.895,C 0.3743,E1 7.8651,E2 193.3548} C_DIS
LIN {X -31.0909,Y -130.8299,Z 174,A -100.2935,B 7.895,C 0.375,E1 7.8691,E2 191.8749} C_DIS
LIN {X -27.4755,Y -131.6377,Z 174,A -98.59,B 7.895,C 0.3737,E1 7.8738,E2 190.1553} C_DIS
LIN {X -23.5254,Y -132.3991,Z 174,A -96.9652,B 7.8949,C 0.3758,E1 7.8782,E2 188.5412} C_DIS
LIN {X -19.5884,Y -133.0398,Z 174,A -95.193,B 7.8949,C 0.3752,E1 7.8832,E2 186.7593} C_DIS
LIN {X -14.5095,Y -133.688,Z 174,A -93.1004,B 7.8949,C 0.3772,E1 7.8889,E2 184.677} C_DIS
LIN {X -11.0853,Y -134.0155,Z 174,A -91.6286,B 7.8949,C 0.3772,E1 7.893,E2 183.2039} C_DIS
LIN {X -7.0776,Y -134.2871,Z 174,A -89.556,B 7.8951,C 0.3711,E1 7.8989,E2 181.085} C_DIS
LIN {X -3.5219,Y -134.4271,Z 174,A -88.0934,B 7.8951,C 0.372,E1 7.903,E2 179.6285} C_DIS
LIN {X -0.1286,Y -134.4745,Z 174,A -87.046,B 7.8948,C 0.3788,E1 7.9058,E2 178.6308} C_DIS
LIN {X -0.1286,Y -134.4745,Z 174,A -87.046,B 7.8948,C 0.3788,E1 7.9058,E2 178.6308} C_DIS
Enddeposition()
LIN {X 0.989,Y -135.3751,Z 174,A -86.4984,B 7.8336,C 0.3827,E1 7.8463,E2 178.1248} C_DIS
Startdeposition()
$VEL.CP = VEL_PRINT
LIN {X -4.5948,Y -135.3035,Z 174,A -89.4877,B 7.8331,C 0.3937,E1 7.8378,E2 181.1943} C_DIS
LIN {X -9.3622,Y -135.0569,Z 174,A -91.5179,B 7.8331,C 0.3937,E1 7.8321,E2 183.2266} C_DIS
LIN {X -13.7953,Y -134.6772,Z 174,A -93.5276,B 7.833,C 0.3956,E1 7.8265,E2 185.2529} C_DIS
LIN {X -18.3201,Y -134.1368,Z 174,A -95.35,B 7.8331,C 0.3934,E1 7.8215,E2 187.0628} C_DIS
LIN {X -22.2045,Y -133.5467,Z 174,A -96.9742,B 7.8331,C 0.3922,E1 7.817,E2 188.6825} C_DIS
LIN {X -26.3145,Y -132.7997,Z 174,A -98.8098,B 7.8331,C 0.3926,E1 7.8119,E2 190.5272} C_DIS
LIN {X -29.9985,Y -132.0145,Z 174,A -100.256,B 7.8333,C 0.3893,E1 7.808,E2 191.9553} C_DIS
LIN {X -33.2623,Y -131.2301,Z 174,A -101.7189,B 7.8333,C 0.3892,E1 7.8041,E2 193.4238} C_DIS
LIN {X -36.4956,Y -130.3679,Z 174,A -103.1531,B 7.8333,C 0.3886,E1 7.8002,E2 194.8606} C_DIS
LIN {X -39.1562,Y -129.5944,Z 174,A -104.9344,B 7.8329,C 0.3976,E1 7.7952,E2 196.718} C_DIS
LIN {X -43.8313,Y -128.089,Z 174,A -106.4895,B 7.8334,C 0.3875,E1 7.7913,E2 198.2084} C_DIS
LIN {X -47.1577,Y -126.9013,Z 174,A -107.7591,B 7.8336,C 0.3826,E1 7.788,E2 199.4499} C_DIS
LIN {X -50.7926,Y -125.4903,Z 174,A -109.5662,B 7.8336,C 0.3835,E1 7.7833,E2 201.2769} C_DIS
LIN {X -53.9418,Y -124.1692,Z 174,A -111.1459,B 7.8336,C 0.3842,E1 7.7792,E2 202.8735} C_DIS
LIN {X -58.0743,Y -122.2911,Z 174,A -112.995,B 7.8337,C 0.3809,E1 7.7745,E2 204.7137} C_DIS
LIN {X -60.944,Y -120.8874,Z 174,A -114.3984,B 7.8337,C 0.3801,E1 7.771,E2 206.1236} C_DIS
LIN {X -64.4066,Y -119.0803,Z 174,A -116.1298,B 7.8338,C 0.3793,E1 7.7667,E2 207.8648} C_DIS
LIN {X -68.3474,Y -116.8627,Z 174,A -118.0482,B 7.8339,C 0.3768,E1 7.762,E2 209.7838} C_DIS
LIN {X -72.1416,Y -114.5591,Z 174,A -119.8723,B 7.8341,C 0.3733,E1 7.7577,E2 211.601} C_DIS
LIN {X -75.2859,Y -112.5178,Z 174,A -121.5431,B 7.8341,C 0.3722,E1 7.7538,E2 213.282} C_DIS
LIN {X -81.0993,Y -108.4029,Z 174,A -124.5811,B 7.8343,C 0.3678,E1 7.7469,E2 216.3226} C_DIS
LIN {X -84.0967,Y -106.0943,Z 174,A -126.4375,B 7.8343,C 0.3689,E1 7.7428,E2 218.2103} C_DIS
LIN {X -86.8061,Y -103.8892,Z 174,A -127.712,B 7.8346,C 0.3632,E1 7.7401,E2 219.4593} C_DIS
LIN {X -90.2357,Y -100.9243,Z 174,A -129.5343,B 7.8348,C 0.3583,E1 7.7363,E2 221.2692} C_DIS
LIN {X -93.5242,Y -97.8847,Z 174,A -131.4919,B 7.8349,C 0.3556,E1 7.7323,E2 223.2341} C_DIS
LIN {X -96.4003,Y -95.0542,Z 174,A -133.3093,B 7.8349,C 0.3539,E1 7.7287,E2 225.0645} C_DIS
LIN {X -100.257,Y -90.9765,Z 174,A -135.4962,B 7.8353,C 0.3463,E1 7.7245,E2 227.2273} C_DIS
LIN {X -102.8431,Y -88.0434,Z 174,A -137.3912,B 7.8353,C 0.3463,E1 7.721,E2 229.1516} C_DIS
LIN {X -105.7266,Y -84.5587,Z 174,A -139.2555,B 7.8355,C 0.3414,E1 7.7177,E2 231.0089} C_DIS
LIN {X -109.6213,Y -79.4441,Z 174,A -141.9617,B 7.8358,C 0.3351,E1 7.7132,E2 233.7122} C_DIS
LIN {X -113.5076,Y -73.785,Z 174,A -145.0196,B 7.836,C 0.3305,E1 7.7084,E2 236.7876} C_DIS
LIN {X -115.9575,Y -69.8721,Z 174,A -146.9788,B 7.8362,C 0.3259,E1 7.7055,E2 238.7465} C_DIS
LIN {X -119.8971,Y -62.8675,Z 174,A -150.3485,B 7.8366,C 0.317,E1 7.701,E2 242.1104} C_DIS
LIN {X -121.3438,Y -60.0279,Z 174,A -151.6212,B 7.8367,C 0.3125,E1 7.6994,E2 243.373} C_DIS
LIN {X -123.4558,Y -55.5555,Z 174,A -153.7811,B 7.8369,C 0.3081,E1 7.6968,E2 245.5399} C_DIS
LIN {X -124.8288,Y -52.3974,Z 174,A -155.3118,B 7.837,C 0.3053,E1 7.6951,E2 247.0787} C_DIS
LIN {X -126.1327,Y -49.1755,Z 174,A -156.8659,B 7.8371,C 0.3025,E1 7.6935,E2 248.642} C_DIS
LIN {X -127.6427,Y -45.1186,Z 174,A -158.8563,B 7.8372,C 0.2998,E1 7.6916,E2 250.6508} C_DIS
LIN {X -128.927,Y -41.298,Z 174,A -160.7739,B 7.8372,C 0.2981,E1 7.6899,E2 252.593} C_DIS
LIN {X -129.9244,Y -38.044,Z 174,A -162.2494,B 7.8374,C 0.2946,E1 7.6887,E2 254.0718} C_DIS
LIN {X -130.8546,Y -34.7105,Z 174,A -163.9116,B 7.8374,C 0.2933,E1 7.6875,E2 255.7569} C_DIS
LIN {X -131.9042,Y -30.4813,Z 174,A -165.2705,B 7.8379,C 0.2815,E1 7.6867,E2 257.0553} C_DIS
LIN {X -132.6211,Y -27.1923,Z 174,A -166.9303,B 7.8379,C 0.2807,E1 7.6857,E2 258.7427} C_DIS
LIN {X -133.4989,Y -22.4905,Z 174,A -168.8143,B 7.8382,C 0.2731,E1 7.6848,E2 260.608} C_DIS
LIN {X -134.0107,Y -19.2065,Z 174,A -170.2129,B 7.8383,C 0.269,E1 7.6843,E2 262.0046} C_DIS
LIN {X -134.4583,Y -15.7731,Z 174,A -171.7416,B 7.8384,C 0.2657,E1 7.6837,E2 263.5398} C_DIS
LIN {X -134.8798,Y -11.6311,Z 174,A -173.6099,B 7.8386,C 0.2621,E1 7.6832,E2 265.4196} C_DIS
LIN {X -135.1949,Y -7.0858,Z 174,A -175.4814,B 7.8388,C 0.2558,E1 7.6829,E2 267.2826} C_DIS
LIN {X -135.3283,Y -3.7498,Z 174,A -176.9787,B 7.8388,C 0.2528,E1 7.6828,E2 268.7889} C_DIS
LIN {X -135.3816,Y 0.4157,Z 174,A -178.8413,B 7.839,C 0.2491,E1 7.6828,E2 270.6621} C_DIS
LIN {X -135.2974,Y 4.7621,Z 174,A 179.3614,B 7.8392,C 0.2432,E1 7.6828,E2 272.4526} C_DIS
LIN {X -135.128,Y 8.2586,Z 174,A 177.8736,B 7.8393,C 0.239,E1 7.6831,E2 273.9398} C_DIS
LIN {X -134.8247,Y 12.269,Z 174,A 176.0429,B 7.8393,C 0.2359,E1 7.6835,E2 275.7846} C_DIS
LIN {X -134.4167,Y 16.122,Z 174,A 174.4304,B 7.8395,C 0.2308,E1 7.684,E2 277.3923} C_DIS
LIN {X -133.8666,Y 20.1932,Z 174,A 172.645,B 7.8397,C 0.2265,E1 7.6847,E2 279.1817} C_DIS
LIN {X -133.3428,Y 23.4016,Z 174,A 171.3337,B 7.8398,C 0.2217,E1 7.6853,E2 280.4839} C_DIS
LIN {X -132.681,Y 26.898,Z 174,A 169.7661,B 7.8399,C 0.2182,E1 7.6862,E2 282.0575} C_DIS
LIN {X -131.9509,Y 30.2772,Z 174,A 168.251,B 7.8399,C 0.2148,E1 7.6871,E2 283.5776} C_DIS
LIN {X -130.9601,Y 34.3147,Z 174,A 166.5258,B 7.8401,C 0.2094,E1 7.6883,E2 285.297} C_DIS
LIN {X -129.9924,Y 37.8119,Z 174,A 164.8845,B 7.8402,C 0.2065,E1 7.6895,E2 286.9495} C_DIS
LIN {X -129.0163,Y 41.0186,Z 174,A 163.4797,B 7.8403,C 0.2024,E1 7.6907,E2 288.3513} C_DIS
LIN {X -127.1322,Y 46.5351,Z 174,A 160.6195,B 7.8403,C 0.201,E1 7.6934,E2 291.2565} C_DIS
LIN {X -125.855,Y 49.8878,Z 174,A 159.2878,B 7.8405,C 0.1944,E1 7.6947,E2 292.5643} C_DIS
LIN {X -124.4057,Y 53.3949,Z 174,A 157.7819,B 7.8407,C 0.1887,E1 7.6964,E2 294.0565} C_DIS
LIN {X -123.0413,Y 56.4681,Z 174,A 156.3541,B 7.8407,C 0.185,E1 7.698,E2 295.4835} C_DIS
LIN {X -121.5445,Y 59.621,Z 174,A 154.8356,B 7.8408,C 0.1817,E1 7.6998,E2 297.0055} C_DIS
LIN {X -119.8349,Y 62.986,Z 174,A 152.5291,B 7.8407,C 0.1873,E1 7.7029,E2 299.3954} C_DIS
LIN {X -117.2375,Y 67.7022,Z 174,A 151.1713,B 7.8411,C 0.169,E1 7.7047,E2 300.6406} C_DIS
LIN {X -114.5336,Y 72.1821,Z 174,A 148.5763,B 7.8411,C 0.1687,E1 7.7085,E2 303.2794} C_DIS
LIN {X -112.1987,Y 75.7606,Z 174,A 147.0385,B 7.8413,C 0.1606,E1 7.7108,E2 304.7828} C_DIS
LIN {X -110.1002,Y 78.7791,Z 174,A 145.1762,B 7.8413,C 0.1612,E1 7.7138,E2 306.6805} C_DIS
LIN {X -107.5487,Y 82.2282,Z 174,A 143.3098,B 7.8413,C 0.1577,E1 7.717,E2 308.5513} C_DIS
LIN {X -104.7552,Y 85.7587,Z 174,A 141.5078,B 7.8415,C 0.1519,E1 7.7201,E2 310.339} C_DIS
LIN {X -102.6384,Y 88.2811,Z 174,A 139.9462,B 7.8415,C 0.1512,E1 7.7229,E2 311.9195} C_DIS
LIN {X -99.9483,Y 91.3155,Z 174,A 138.0434,B 7.8415,C 0.1501,E1 7.7265,E2 313.843} C_DIS
LIN {X -96.3313,Y 95.1244,Z 174,A 136.0021,B 7.8416,C 0.1429,E1 7.7305,E2 315.8605} C_DIS
LIN {X -92.939,Y 98.4406,Z 174,A 134.0923,B 7.8417,C 0.1375,E1 7.7343,E2 317.7567} C_DIS
LIN {X -91.1794,Y 100.0729,Z 174,A 132.4839,B 7.8417,C 0.1439,E1 7.7378,E2 319.435} C_DIS
LIN {X -87.9525,Y 102.9207,Z 174,A 130.9998,B 7.8417,C 0.1357,E1 7.7408,E2 320.8773} C_DIS
LIN {X -84.3769,Y 105.8713,Z 174,A 129.0657,B 7.8418,C 0.1317,E1 7.745,E2 322.8062} C_DIS
LIN {X -81.0523,Y 108.4379,Z 174,A 127.4293,B 7.8419,C 0.1265,E1 7.7486,E2 324.4242} C_DIS
LIN {X -76.175,Y 111.9182,Z 174,A 124.6591,B 7.8419,C 0.1257,E1 7.755,E2 327.2203} C_DIS
LIN {X -72.404,Y 114.3936,Z 174,A 122.8712,B 7.8419,C 0.1209,E1 7.7591,E2 328.9921} C_DIS
LIN {X -69.3891,Y 116.2469,Z 174,A 120.8831,B 7.8419,C 0.1259,E1 7.764,E2 331.0373} C_DIS
LIN {X -65.8035,Y 118.3138,Z 174,A 119.5995,B 7.8421,C 0.1165,E1 7.767,E2 332.2638} C_DIS
LIN {X -62.3521,Y 120.1675,Z 174,A 117.1648,B 7.8419,C 0.1258,E1 7.7733,E2 334.7894} C_DIS
LIN {X -57.3527,Y 122.6322,Z 174,A 115.5607,B 7.8421,C 0.1115,E1 7.7771,E2 336.302} C_DIS
LIN {X -54.0232,Y 124.134,Z 174,A 113.9559,B 7.8421,C 0.1106,E1 7.7812,E2 337.9127} C_DIS
LIN {X -50.8316,Y 125.4746,Z 174,A 111.5999,B 7.842,C 0.1225,E1 7.7876,E2 340.3734} C_DIS
LIN {X -44.8264,Y 127.744,Z 174,A 109.7344,B 7.8422,C 0.1069,E1 7.7922,E2 342.136} C_DIS
LIN {X -41.4743,Y 128.8707,Z 174,A 108.2588,B 7.8422,C 0.1052,E1 7.7961,E2 343.608} C_DIS
LIN {X -34.7556,Y 130.8425,Z 174,A 105.2161,B 7.8422,C 0.104,E1 7.8043,E2 346.6583} C_DIS
LIN {X -30.4303,Y 131.9159,Z 174,A 103.3532,B 7.8422,C 0.1024,E1 7.8093,E2 348.5172} C_DIS
LIN {X -27.0793,Y 132.6441,Z 174,A 101.9606,B 7.8422,C 0.1006,E1 7.8131,E2 349.9019} C_DIS
LIN {X -23.9262,Y 133.2489,Z 174,A 100.5652,B 7.8422,C 0.1004,E1 7.8169,E2 351.3008} C_DIS
LIN {X -20.7144,Y 133.7859,Z 174,A 99.1794,B 7.8422,C 0.0999,E1 7.8208,E2 352.6867} C_DIS
LIN {X -17.091,Y 134.2978,Z 174,A 97.4968,B 7.8422,C 0.1015,E1 7.8255,E2 354.3846} C_DIS
LIN {X -13.0014,Y 134.7544,Z 174,A 95.8643,B 7.8422,C 0.0992,E1 7.83,E2 356.003} C_DIS
LIN {X -9.1606,Y 135.0717,Z 174,A 94.1282,B 7.8422,C 0.1005,E1 7.8348,E2 357.7509} C_DIS
LIN {X -5.1717,Y 135.2814,Z 174,A 92.517,B 7.8423,C 0.099,E1 7.8393,E2 359.3518} C_DIS
LIN {X -0.9145,Y 135.3773,Z 174,A 90.9248,B 7.8423,C 0.0955,E1 7.8437,E2 360.9179} C_DIS
LIN {X 2.8447,Y 135.3516,Z 174,A 89.0371,B 7.8423,C 0.1004,E1 7.849,E2 362.8405} C_DIS
LIN {X 6.9595,Y 135.2013,Z 174,A 87.3586,B 7.8423,C 0.0996,E1 7.8537,E2 364.5106} C_DIS
LIN {X 11.0629,Y 134.9278,Z 174,A 85.6273,B 7.8423,C 0.0998,E1 7.8585,E2 366.2401} C_DIS
LIN {X 14.7685,Y 134.5724,Z 174,A 84.004,B 7.8423,C 0.101,E1 7.863,E2 367.8686} C_DIS
LIN {X 19.0089,Y 134.0389,Z 174,A 82.2916,B 7.8423,C 0.1001,E1 7.8677,E2 369.5689} C_DIS
LIN {X 22.5681,Y 133.486,Z 174,A 80.7641,B 7.8423,C 0.1008,E1 7.872,E2 371.0963} C_DIS
LIN {X 26.4529,Y 132.7715,Z 174,A 79.0403,B 7.8423,C 0.1026,E1 7.8767,E2 372.8259} C_DIS
LIN {X 29.9077,Y 132.0353,Z 174,A 77.6059,B 7.8423,C 0.1025,E1 7.8806,E2 374.2526} C_DIS
LIN {X 33.2026,Y 131.2452,Z 174,A 76.1944,B 7.8423,C 0.1031,E1 7.8844,E2 375.6611} C_DIS
LIN {X 36.4038,Y 130.3935,Z 174,A 74.1757,B 7.8421,C 0.1148,E1 7.8901,E2 377.7531} C_DIS
LIN {X 41.2284,Y 128.9493,Z 174,A 72.6984,B 7.8422,C 0.1053,E1 7.8938,E2 379.1519} C_DIS
LIN {X 44.0948,Y 127.9977,Z 174,A 71.5677,B 7.8422,C 0.1039,E1 7.8967,E2 380.2647} C_DIS
LIN {X 47.4896,Y 126.777,Z 174,A 69.8751,B 7.8422,C 0.1083,E1 7.9012,E2 381.9771} C_DIS
LIN {X 50.726,Y 125.5171,Z 174,A 68.35,B 7.8422,C 0.1108,E1 7.9052,E2 383.5087} C_DIS
LIN {X 55.0954,Y 123.6616,Z 174,A 66.4605,B 7.8422,C 0.111,E1 7.91,E2 385.3837} C_DIS
LIN {X 57.9135,Y 122.368,Z 174,A 65.1053,B 7.8422,C 0.1133,E1 7.9134,E2 386.744} C_DIS
LIN {X 61.2418,Y 120.7357,Z 174,A 63.6044,B 7.8421,C 0.1141,E1 7.9172,E2 388.2366} C_DIS
LIN {X 64.4591,Y 119.0521,Z 174,A 61.9379,B 7.8421,C 0.1185,E1 7.9213,E2 389.9189} C_DIS
LIN {X 68.356,Y 116.8577,Z 174,A 60.0738,B 7.842,C 0.1207,E1 7.9258,E2 391.7796} C_DIS
LIN {X 72.2338,Y 114.5009,Z 174,A 58.1885,B 7.842,C 0.1229,E1 7.9303,E2 393.6608} C_DIS
LIN {X 77.1212,Y 111.268,Z 174,A 55.72,B 7.842,C 0.1267,E1 7.936,E2 396.1281} C_DIS
LIN {X 80.7915,Y 108.6321,Z 174,A 53.8378,B 7.8419,C 0.1294,E1 7.9402,E2 398.007} C_DIS
LIN {X 84.5219,Y 105.7559,Z 174,A 51.8638,B 7.8419,C 0.1325,E1 7.9446,E2 399.9789} C_DIS
LIN {X 88.0345,Y 102.8508,Z 174,A 50.0544,B 7.8418,C 0.1338,E1 7.9484,E2 401.7742} C_DIS
LIN {X 91.0703,Y 100.1719,Z 174,A 48.3041,B 7.8418,C 0.1378,E1 7.9521,E2 403.5294} C_DIS
LIN {X 94.1718,Y 97.2619,Z 174,A 46.5154,B 7.8417,C 0.1411,E1 7.9557,E2 405.3173} C_DIS
LIN {X 97.5623,Y 93.8613,Z 174,A 44.4518,B 7.8416,C 0.1459,E1 7.9597,E2 407.3853} C_DIS
LIN {X 100.6381,Y 90.5553,Z 174,A 42.5734,B 7.8416,C 0.1493,E1 7.9633,E2 409.2604} C_DIS
LIN {X 103.5514,Y 87.2087,Z 174,A 40.9496,B 7.8416,C 0.1486,E1 7.9662,E2 410.854} C_DIS
LIN {X 107.1303,Y 82.7728,Z 174,A 38.3787,B 7.8414,C 0.157,E1 7.9707,E2 413.4452} C_DIS
LIN {X 109.7416,Y 79.2781,Z 174,A 36.6332,B 7.8414,C 0.1593,E1 7.9735,E2 415.1792} C_DIS
LIN {X 112.159,Y 75.8193,Z 174,A 34.8121,B 7.8412,C 0.1642,E1 7.9764,E2 417.0054} C_DIS
LIN {X 114.6567,Y 71.9871,Z 174,A 32.9574,B 7.8412,C 0.1673,E1 7.9792,E2 418.8511} C_DIS
LIN {X 116.8213,Y 68.418,Z 174,A 31.1564,B 7.841,C 0.1723,E1 7.9818,E2 420.6573} C_DIS
LIN {X 119.0498,Y 64.4633,Z 174,A 29.2165,B 7.841,C 0.1775,E1 7.9844,E2 422.6005} C_DIS
LIN {X 121.1182,Y 60.4853,Z 174,A 27.4597,B 7.8409,C 0.1796,E1 7.9866,E2 424.3411} C_DIS
LIN {X 122.7581,Y 57.0806,Z 174,A 25.8847,B 7.8408,C 0.1833,E1 7.9885,E2 425.9141} C_DIS
LIN {X 124.1238,Y 54.0468,Z 174,A 24.4882,B 7.8408,C 0.1867,E1 7.9901,E2 427.31} C_DIS
LIN {X 125.7526,Y 50.1419,Z 174,A 22.4754,B 7.8405,C 0.1958,E1 7.9922,E2 429.3511} C_DIS
LIN {X 126.9315,Y 47.0771,Z 174,A 21.1794,B 7.8405,C 0.1978,E1 7.9935,E2 430.6366} C_DIS
LIN {X 128.3839,Y 42.957,Z 174,A 19.6568,B 7.8405,C 0.1964,E1 7.9948,E2 432.1204} C_DIS
LIN {X 129.7596,Y 38.6068,Z 174,A 17.5978,B 7.8403,C 0.2042,E1 7.9966,E2 434.1966} C_DIS
LIN {X 130.72,Y 35.215,Z 174,A 16.2067,B 7.8403,C 0.2063,E1 7.9976,E2 435.5763} C_DIS
LIN {X 131.5848,Y 31.8303,Z 174,A 14.7831,B 7.8401,C 0.2094,E1 7.9985,E2 436.9943} C_DIS
LIN {X 132.3374,Y 28.5403,Z 174,A 13.3866,B 7.8401,C 0.2127,E1 7.9994,E2 438.3879} C_DIS
LIN {X 132.9749,Y 25.4052,Z 174,A 12.0261,B 7.8399,C 0.2167,E1 8.0001,E2 439.7503} C_DIS
LIN {X 133.6626,Y 21.5097,Z 174,A 10.2804,B 7.8398,C 0.2229,E1 8.0009,E2 441.5061} C_DIS
LIN {X 134.2203,Y 17.6825,Z 174,A 8.8068,B 7.8398,C 0.2243,E1 8.0015,E2 442.9609} C_DIS
LIN {X 134.5729,Y 14.7641,Z 174,A 7.5296,B 7.8396,C 0.2285,E1 8.0019,E2 444.2432} C_DIS
LIN {X 134.9327,Y 11.0045,Z 174,A 5.9034,B 7.8395,C 0.2336,E1 8.0023,E2 445.8742} C_DIS
LIN {X 135.205,Y 6.8857,Z 174,A 4.4457,B 7.8395,C 0.2329,E1 8.0025,E2 447.2975} C_DIS
LIN {X 135.3455,Y 3.131,Z 174,A 2.6012,B 7.8392,C 0.2426,E1 8.0027,E2 449.175} C_DIS
LIN {X 135.3793,Y -0.7505,Z 174,A 1.0553,B 7.8392,C 0.2454,E1 8.0027,E2 450.7103} C_DIS
LIN {X 135.2904,Y -4.9408,Z 174,A -0.5165,B 7.8391,C 0.2465,E1 8.0027,E2 452.2586} C_DIS
LIN {X 135.168,Y -7.5934,Z 174,A -2.2782,B 7.8386,C 0.2624,E1 8.0023,E2 454.1001} C_DIS
LIN {X 134.8239,Y -12.2767,Z 174,A -3.747,B 7.8387,C 0.2578,E1 8.002,E2 455.5068} C_DIS
LIN {X 134.4801,Y -15.5908,Z 174,A -5.0685,B 7.8387,C 0.2601,E1 8.0016,E2 456.8187} C_DIS
LIN {X 134.0612,Y -18.853,Z 174,A -6.4761,B 7.8385,C 0.2644,E1 8.001,E2 458.2294} C_DIS
LIN {X 133.5571,Y -22.1417,Z 174,A -7.7656,B 7.8385,C 0.2661,E1 8.0005,E2 459.5055} C_DIS
LIN {X 132.983,Y -25.3626,Z 174,A -9.0753,B 7.8384,C 0.2685,E1 7.9998,E2 460.8073} C_DIS
LIN {X 132.3706,Y -28.3862,Z 174,A -10.4012,B 7.8382,C 0.2726,E1 7.9991,E2 462.137} C_DIS
LIN {X 131.7202,Y -31.2686,Z 174,A -12.3925,B 7.8376,C 0.2909,E1 7.9977,E2 464.2211} C_DIS
LIN {X 130.3425,Y -36.5862,Z 174,A -14.0241,B 7.8378,C 0.2837,E1 7.9966,E2 465.7692} C_DIS
LIN {X 129.0744,Y -40.8368,Z 174,A -15.8069,B 7.8378,C 0.287,E1 7.9951,E2 467.5422} C_DIS
LIN {X 127.9726,Y -44.1671,Z 174,A -17.026,B 7.8378,C 0.2858,E1 7.9941,E2 468.7295} C_DIS
LIN {X 126.9408,Y -47.0522,Z 174,A -18.5909,B 7.8374,C 0.2947,E1 7.9926,E2 470.3293} C_DIS
LIN {X 125.6849,Y -50.3099,Z 174,A -20.037,B 7.8373,C 0.2981,E1 7.9911,E2 471.7728} C_DIS
LIN {X 124.1238,Y -54.0468,Z 174,A -22.384,B 7.8366,C 0.3152,E1 7.9884,E2 474.2} C_DIS
LIN {X 121.7835,Y -59.1363,Z 174,A -24.1023,B 7.8369,C 0.3086,E1 7.9864,E2 475.8399} C_DIS
LIN {X 120.0418,Y -62.592,Z 174,A -25.6353,B 7.8368,C 0.3108,E1 7.9845,E2 477.3614} C_DIS
LIN {X 118.4054,Y -65.6382,Z 174,A -27.3981,B 7.8364,C 0.3205,E1 7.9821,E2 479.163} C_DIS
LIN {X 116.6551,Y -68.7009,Z 174,A -28.5807,B 7.8365,C 0.3182,E1 7.9805,E2 480.3085} C_DIS
LIN {X 114.4378,Y -72.3339,Z 174,A -30.3939,B 7.8363,C 0.3229,E1 7.9778,E2 482.125} C_DIS
LIN {X 111.9087,Y -76.189,Z 174,A -32.628,B 7.8359,C 0.3332,E1 7.9742,E2 484.3962} C_DIS
LIN {X 109.6912,Y -79.3477,Z 174,A -33.9173,B 7.836,C 0.3304,E1 7.9722,E2 485.6443} C_DIS
LIN {X 107.8761,Y -81.7987,Z 174,A -35.3059,B 7.8358,C 0.3354,E1 7.9698,E2 487.0464} C_DIS
LIN {X 104.6846,Y -85.8451,Z 174,A -37.5418,B 7.8355,C 0.3415,E1 7.9659,E2 489.2913} C_DIS
LIN {X 102.5903,Y -88.337,Z 174,A -38.6697,B 7.8356,C 0.3398,E1 7.9639,E2 490.3893} C_DIS
LIN {X 99.8498,Y -91.4236,Z 174,A -40.4461,B 7.8354,C 0.3442,E1 7.9606,E2 492.1711} C_DIS
LIN {X 96.8296,Y -94.6165,Z 174,A -42.1246,B 7.8354,C 0.3447,E1 7.9574,E2 493.8286} C_DIS
LIN {X 93.6883,Y -97.7278,Z 174,A -44.0922,B 7.8351,C 0.3505,E1 7.9534,E2 495.8101} C_DIS
LIN {X 90.5965,Y -100.6012,Z 174,A -45.8358,B 7.8351,C 0.3533,E1 7.9498,E2 497.5501} C_DIS
LIN {X 87.4102,Y -103.3817,Z 174,A -47.6575,B 7.8348,C 0.3574,E1 7.946,E2 499.3775} C_DIS
LIN {X 84.8822,Y -105.4667,Z 174,A -49.2803,B 7.8345,C 0.3645,E1 7.9424,E2 501.031} C_DIS
LIN {X 81.9534,Y -107.7589,Z 174,A -50.5472,B 7.8346,C 0.3616,E1 7.9396,E2 502.261} C_DIS
LIN {X 78.5866,Y -110.2378,Z 174,A -52.3513,B 7.8345,C 0.3654,E1 7.9356,E2 504.071} C_DIS
LIN {X 74.7219,Y -112.8935,Z 174,A -54.3052,B 7.8343,C 0.3682,E1 7.931,E2 506.0228} C_DIS
LIN {X 71.318,Y -115.0739,Z 174,A -55.8104,B 7.8343,C 0.3671,E1 7.9275,E2 507.5036} C_DIS
LIN {X 68.7339,Y -116.6357,Z 174,A -57.2027,B 7.8342,C 0.3713,E1 7.9242,E2 508.9114} C_DIS
LIN {X 63.1918,Y -119.7269,Z 174,A -59.8122,B 7.8341,C 0.3738,E1 7.9178,E2 511.5135} C_DIS
LIN {X 60.16,Y -121.2786,Z 174,A -61.2742,B 7.8339,C 0.3762,E1 7.9141,E2 512.9793} C_DIS
LIN {X 57.5081,Y -122.5604,Z 174,A -62.5139,B 7.8339,C 0.3778,E1 7.911,E2 514.2192} C_DIS
LIN {X 54.3796,Y -123.9799,Z 174,A -64.0243,B 7.8337,C 0.3807,E1 7.9071,E2 515.7378} C_DIS
LIN {X 50.8473,Y -125.4682,Z 174,A -65.4259,B 7.8338,C 0.3786,E1 7.9036,E2 517.1129} C_DIS
LIN {X 48.0601,Y -126.5633,Z 174,A -66.833,B 7.8336,C 0.3826,E1 7.8999,E2 518.5386} C_DIS
LIN {X 44.5333,Y -127.8456,Z 174,A -68.3212,B 7.8336,C 0.3826,E1 7.896,E2 520.0154} C_DIS
LIN {X 41.5827,Y -128.8361,Z 174,A -69.6948,B 7.8336,C 0.3849,E1 7.8923,E2 521.3971} C_DIS
LIN {X 38.1955,Y -129.88,Z 174,A -71.11,B 7.8336,C 0.3847,E1 7.8886,E2 522.8026} C_DIS
LIN {X 35.1071,Y -130.7488,Z 174,A -72.4525,B 7.8335,C 0.3857,E1 7.8849,E2 524.1441} C_DIS
LIN {X 31.8499,Y -131.5801,Z 174,A -73.9243,B 7.8334,C 0.3877,E1 7.8809,E2 525.6231} C_DIS
LIN {X 28.4337,Y -132.3604,Z 174,A -75.4265,B 7.8334,C 0.3891,E1 7.8768,E2 527.1287} C_DIS
LIN {X 24.1692,Y -133.2055,Z 174,A -77.2178,B 7.8334,C 0.3895,E1 7.8719,E2 528.915} C_DIS
LIN {X 21.0094,Y -133.7402,Z 174,A -78.6859,B 7.8332,C 0.3923,E1 7.8678,E2 530.398} C_DIS
LIN {X 16.3583,Y -134.3885,Z 174,A -80.5508,B 7.8332,C 0.3911,E1 7.8627,E2 532.2487} C_DIS
LIN {X 9.6311,Y -135.0373,Z 174,A -83.3211,B 7.8332,C 0.3906,E1 7.8551,E2 535.0093} C_DIS
LIN {X 2.9271,Y -135.3503,Z 174,A -86.3694,B 7.833,C 0.3949,E1 7.8465,E2 538.0853} C_DIS
LIN {X 2.9271,Y -135.3503,Z 174,A -86.3694,B 7.833,C 0.3949,E1 7.8465,E2 538.0853} C_DIS
Enddeposition()
LIN {X 0.9737,Y -136.2785,Z 174,A -87.9431,B 7.8149,C 0.4126,E1 7.8246,E2 539.7918} C_DIS
Startdeposition()
$VEL.CP = VEL_PRINT
LIN {X 8.4641,Y -136.0242,Z 174,A -82.309,B 7.8171,C 0.3685,E1 7.8411,E2 533.8405} C_DIS
LIN {X 15.2725,Y -135.4306,Z 174,A -80.4065,B 7.8163,C 0.3848,E1 7.8461,E2 532.0619} C_DIS
LIN {X 19.9,Y -134.8279,Z 174,A -78.372,B 7.8164,C 0.3825,E1 7.8517,E2 530.017} C_DIS
LIN {X 23.7713,Y -134.1982,Z 174,A -76.7346,B 7.8164,C 0.3817,E1 7.8562,E2 528.38} C_DIS
LIN {X 27.5935,Y -133.4652,Z 174,A -75.1913,B 7.8164,C 0.3822,E1 7.8604,E2 526.8476} C_DIS
LIN {X 30.4294,Y -132.8466,Z 174,A -73.9357,B 7.8165,C 0.3807,E1 7.8639,E2 525.5867} C_DIS
LIN {X 33.6963,Y -132.0558,Z 174,A -72.5226,B 7.8165,C 0.3795,E1 7.8677,E2 524.1726} C_DIS
LIN {X 37.3989,Y -131.0572,Z 174,A -70.8173,B 7.8167,C 0.3764,E1 7.8723,E2 522.4543} C_DIS
LIN {X 41.2741,Y -129.8869,Z 174,A -69.1835,B 7.8167,C 0.376,E1 7.8766,E2 520.828} C_DIS
LIN {X 44.6375,Y -128.7696,Z 174,A -67.7279,B 7.8168,C 0.3751,E1 7.8805,E2 519.3756} C_DIS
LIN {X 47.7642,Y -127.6428,Z 174,A -66.3482,B 7.8168,C 0.3739,E1 7.8841,E2 517.9972} C_DIS
LIN {X 51.1173,Y -126.3374,Z 174,A -64.8452,B 7.8169,C 0.3723,E1 7.888,E2 516.4943} C_DIS
LIN {X 54.32,Y -124.994,Z 174,A -63.4024,B 7.817,C 0.3708,E1 7.8917,E2 515.0525} C_DIS
LIN {X 58.0373,Y -123.3142,Z 174,A -61.7481,B 7.817,C 0.3697,E1 7.8959,E2 513.4047} C_DIS
LIN {X 61.0289,Y -121.8615,Z 174,A -60.3407,B 7.8172,C 0.3676,E1 7.8994,E2 511.995} C_DIS
LIN {X 63.9675,Y -120.3441,Z 174,A -58.1944,B 7.8179,C 0.3511,E1 7.905,E2 509.75} C_DIS
LIN {X 69.1028,Y -117.471,Z 174,A -56.7361,B 7.8172,C 0.3668,E1 7.9082,E2 508.4204} C_DIS
LIN {X 72.4629,Y -115.4291,Z 174,A -54.752,B 7.8176,C 0.3578,E1 7.913,E2 506.3926} C_DIS
LIN {X 76.2424,Y -112.9679,Z 174,A -52.8902,B 7.8177,C 0.3552,E1 7.9173,E2 504.5335} C_DIS
LIN {X 79.9922,Y -110.3444,Z 174,A -51.0229,B 7.8178,C 0.3529,E1 7.9215,E2 502.6717} C_DIS
LIN {X 83.5326,Y -107.6891,Z 174,A -49.1033,B 7.818,C 0.3484,E1 7.9258,E2 500.7429} C_DIS
LIN {X 87.2908,Y -104.6667,Z 174,A -47.13,B 7.8182,C 0.3456,E1 7.9301,E2 498.7747} C_DIS
LIN {X 90.2729,Y -102.105,Z 174,A -45.5611,B 7.8182,C 0.3439,E1 7.9334,E2 497.215} C_DIS
LIN {X 93.3995,Y -99.2531,Z 174,A -43.7914,B 7.8184,C 0.3405,E1 7.937,E2 495.4448} C_DIS
LIN {X 96.4921,Y -96.2496,Z 174,A -41.9715,B 7.8185,C 0.3365,E1 7.9406,E2 493.6222} C_DIS
LIN {X 99.5562,Y -93.0766,Z 174,A -40.1737,B 7.8187,C 0.3336,E1 7.944,E2 491.8299} C_DIS
LIN {X 102.39,Y -89.9504,Z 174,A -38.4185,B 7.8188,C 0.33,E1 7.9473,E2 490.0754} C_DIS
LIN {X 105.0592,Y -86.8171,Z 174,A -36.8395,B 7.8188,C 0.3291,E1 7.9501,E2 488.514} C_DIS
LIN {X 107.4671,Y -83.819,Z 174,A -35.2227,B 7.819,C 0.3254,E1 7.9529,E2 486.8956} C_DIS
LIN {X 109.6736,Y -80.9099,Z 174,A -33.6175,B 7.8192,C 0.3203,E1 7.9556,E2 485.28} C_DIS
LIN {X 112.1849,Y -77.3905,Z 174,A -31.9145,B 7.8193,C 0.3182,E1 7.9583,E2 483.5898} C_DIS
LIN {X 114.2516,Y -74.3049,Z 174,A -29.9904,B 7.8198,C 0.3071,E1 7.9614,E2 481.6177} C_DIS
LIN {X 116.2595,Y -71.1221,Z 174,A -28.8625,B 7.8195,C 0.3122,E1 7.9629,E2 480.5463} C_DIS
LIN {X 118.2019,Y -67.846,Z 174,A -27.2806,B 7.8197,C 0.3086,E1 7.9652,E2 478.9653} C_DIS
LIN {X 119.9417,Y -64.7201,Z 174,A -25.6533,B 7.8199,C 0.3022,E1 7.9674,E2 477.3208} C_DIS
LIN {X 121.8061,Y -61.1386,Z 174,A -24.0617,B 7.82,C 0.2999,E1 7.9694,E2 475.7409} C_DIS
LIN {X 123.562,Y -57.5033,Z 174,A -22.1716,B 7.8203,C 0.2915,E1 7.9716,E2 473.8245} C_DIS
LIN {X 125.7875,Y -52.4558,Z 174,A -20.148,B 7.8203,C 0.2913,E1 7.9738,E2 471.8363} C_DIS
LIN {X 127.0851,Y -49.2292,Z 174,A -18.678,B 7.8205,C 0.2871,E1 7.9754,E2 470.3639} C_DIS
LIN {X 128.4549,Y -45.5408,Z 174,A -17.0952,B 7.8206,C 0.2841,E1 7.9769,E2 468.7886} C_DIS
LIN {X 129.4968,Y -42.4861,Z 174,A -15.7748,B 7.8207,C 0.281,E1 7.978,E2 467.4714} C_DIS
LIN {X 130.454,Y -39.4472,Z 174,A -14.4177,B 7.8209,C 0.277,E1 7.9791,E2 466.1108} C_DIS
LIN {X 131.5086,Y -35.7786,Z 174,A -12.5411,B 7.8212,C 0.2669,E1 7.9806,E2 464.1981} C_DIS
LIN {X 132.3546,Y -32.5076,Z 174,A -11.557,B 7.821,C 0.2718,E1 7.9812,E2 463.268} C_DIS
LIN {X 133.2935,Y -28.4102,Z 174,A -9.7369,B 7.8213,C 0.2657,E1 7.9823,E2 461.4395} C_DIS
LIN {X 134.0371,Y -24.6713,Z 174,A -8.0772,B 7.8214,C 0.26,E1 7.9832,E2 459.7711} C_DIS
LIN {X 134.6824,Y -20.853,Z 174,A -6.6016,B 7.8215,C 0.2584,E1 7.9838,E2 458.3132} C_DIS
LIN {X 135.1601,Y -17.4923,Z 174,A -5.1728,B 7.8216,C 0.2543,E1 7.9844,E2 456.8828} C_DIS
LIN {X 135.5661,Y -14.0132,Z 174,A -3.4995,B 7.8219,C 0.246,E1 7.9849,E2 455.1828} C_DIS
LIN {X 136.0744,Y -7.6385,Z 174,A -0.6957,B 7.8222,C 0.2359,E1 7.9854,E2 452.362} C_DIS
LIN {X 136.2291,Y -3.9905,Z 174,A 0.4112,B 7.8221,C 0.2402,E1 7.9855,E2 451.3079} C_DIS
LIN {X 136.2891,Y -0.3555,Z 174,A 2.1267,B 7.8223,C 0.232,E1 7.9855,E2 449.5675} C_DIS
LIN {X 136.2222,Y 4.2361,Z 174,A 3.7865,B 7.8223,C 0.2319,E1 7.9855,E2 447.9401} C_DIS
LIN {X 136.1176,Y 6.7999,Z 174,A 4.967,B 7.8225,C 0.2267,E1 7.9853,E2 446.7458} C_DIS
LIN {X 135.8237,Y 11.2339,Z 174,A 6.7439,B 7.8225,C 0.2232,E1 7.9849,E2 444.979} C_DIS
LIN {X 135.4783,Y 14.8294,Z 174,A 8.2293,B 7.8227,C 0.2195,E1 7.9845,E2 443.4964} C_DIS
LIN {X 135.0101,Y 18.6252,Z 174,A 9.8717,B 7.8228,C 0.2142,E1 7.9839,E2 441.8484} C_DIS
LIN {X 134.401,Y 22.5962,Z 174,A 11.4639,B 7.8229,C 0.2114,E1 7.9832,E2 440.2671} C_DIS
LIN {X 133.6335,Y 26.766,Z 174,A 13.2518,B 7.823,C 0.2062,E1 7.9823,E2 438.477} C_DIS
LIN {X 132.7985,Y 30.6397,Z 174,A 14.8467,B 7.8231,C 0.203,E1 7.9813,E2 436.8898} C_DIS
LIN {X 132.0659,Y 33.6565,Z 174,A 16.1269,B 7.8232,C 0.1998,E1 7.9804,E2 435.6118} C_DIS
LIN {X 131.2218,Y 36.8103,Z 174,A 17.4831,B 7.8232,C 0.1964,E1 7.9794,E2 434.2566} C_DIS
LIN {X 130.1429,Y 40.4638,Z 174,A 19.0454,B 7.8234,C 0.1928,E1 7.9782,E2 432.6982} C_DIS
LIN {X 129.1355,Y 43.5711,Z 174,A 20.4782,B 7.8235,C 0.1878,E1 7.9769,E2 431.257} C_DIS
LIN {X 127.0163,Y 49.406,Z 174,A 22.7996,B 7.8235,C 0.1866,E1 7.9747,E2 428.9699} C_DIS
LIN {X 125.67,Y 52.7371,Z 174,A 24.4675,B 7.8237,C 0.1794,E1 7.9729,E2 427.2814} C_DIS
LIN {X 124.3099,Y 55.8676,Z 174,A 25.8838,B 7.8237,C 0.176,E1 7.9713,E2 425.8665} C_DIS
LIN {X 122.8187,Y 59.0743,Z 174,A 27.3252,B 7.8238,C 0.1731,E1 7.9696,E2 424.43} C_DIS
LIN {X 121.342,Y 62.0504,Z 174,A 28.6856,B 7.8239,C 0.1702,E1 7.9679,E2 423.0733} C_DIS
LIN {X 119.6717,Y 65.2176,Z 174,A 30.2667,B 7.824,C 0.1649,E1 7.9658,E2 421.482} C_DIS
LIN {X 117.3672,Y 69.2796,Z 174,A 32.2003,B 7.8241,C 0.1606,E1 7.9631,E2 419.5511} C_DIS
LIN {X 115.0479,Y 73.0668,Z 174,A 34.0679,B 7.8241,C 0.1561,E1 7.9603,E2 417.6825} C_DIS
LIN {X 112.5951,Y 76.7928,Z 174,A 35.9177,B 7.8243,C 0.1521,E1 7.9574,E2 415.835} C_DIS
LIN {X 109.9094,Y 80.5889,Z 174,A 37.8137,B 7.8243,C 0.1487,E1 7.9543,E2 413.9454} C_DIS
LIN {X 107.0994,Y 84.2874,Z 174,A 39.8345,B 7.8244,C 0.143,E1 7.9509,E2 411.9154} C_DIS
LIN {X 103.9832,Y 88.1033,Z 174,A 41.7897,B 7.8244,C 0.1407,E1 7.9474,E2 409.9738} C_DIS
LIN {X 101.072,Y 91.4282,Z 174,A 43.6281,B 7.8245,C 0.1371,E1 7.944,E2 408.1372} C_DIS
LIN {X 98.0009,Y 94.7125,Z 174,A 45.4678,B 7.8245,C 0.1341,E1 7.9404,E2 406.3032} C_DIS
LIN {X 95.0183,Y 97.7049,Z 174,A 47.2575,B 7.8247,C 0.1303,E1 7.9369,E2 404.5113} C_DIS
LIN {X 91.7336,Y 100.7949,Z 174,A 49.0553,B 7.8247,C 0.1285,E1 7.9332,E2 402.7252} C_DIS
LIN {X 88.9636,Y 103.2478,Z 174,A 50.6219,B 7.8247,C 0.1254,E1 7.9299,E2 401.1568} C_DIS
LIN {X 85.5332,Y 106.107,Z 174,A 52.4906,B 7.8247,C 0.1221,E1 7.9259,E2 399.2888} C_DIS
LIN {X 81.8906,Y 108.9432,Z 174,A 54.4126,B 7.8248,C 0.1191,E1 7.9216,E2 397.3688} C_DIS
LIN {X 78.2182,Y 111.6096,Z 174,A 56.2718,B 7.8248,C 0.1168,E1 7.9174,E2 395.5154} C_DIS
LIN {X 74.5361,Y 114.1015,Z 174,A 58.1774,B 7.8249,C 0.1132,E1 7.913,E2 393.6052} C_DIS
LIN {X 70.7805,Y 116.4682,Z 174,A 60.0133,B 7.8249,C 0.111,E1 7.9086,E2 391.7728} C_DIS
LIN {X 66.9379,Y 118.7181,Z 174,A 61.8624,B 7.8249,C 0.1087,E1 7.9041,E2 389.9264} C_DIS
LIN {X 63.0079,Y 120.848,Z 174,A 63.6404,B 7.825,C 0.108,E1 7.8998,E2 388.1609} C_DIS
LIN {X 59.9983,Y 122.3699,Z 174,A 65.0403,B 7.825,C 0.1065,E1 7.8963,E2 386.7632} C_DIS
LIN {X 57.0238,Y 123.7837,Z 174,A 66.4211,B 7.825,C 0.1049,E1 7.8928,E2 385.3829} C_DIS
LIN {X 53.1384,Y 125.5024,Z 174,A 68.5872,B 7.8252,C 0.0961,E1 7.8871,E2 383.1701} C_DIS
LIN {X 49.577,Y 126.9499,Z 174,A 69.5379,B 7.825,C 0.1063,E1 7.8849,E2 382.3015} C_DIS
LIN {X 45.9041,Y 128.324,Z 174,A 71.3985,B 7.825,C 0.1009,E1 7.8799,E2 380.4151} C_DIS
LIN {X 42.7268,Y 129.4166,Z 174,A 72.8414,B 7.8251,C 0.0991,E1 7.8761,E2 378.9687} C_DIS
LIN {X 38.307,Y 130.7926,Z 174,A 74.7861,B 7.8251,C 0.0975,E1 7.8709,E2 377.0245} C_DIS
LIN {X 35.0107,Y 131.7133,Z 174,A 76.1766,B 7.8251,C 0.0972,E1 7.8672,E2 375.6402} C_DIS
LIN {X 31.6657,Y 132.5576,Z 174,A 77.6974,B 7.8251,C 0.095,E1 7.863,E2 374.1112} C_DIS
LIN {X 27.529,Y 133.4783,Z 174,A 79.448,B 7.8251,C 0.0945,E1 7.8583,E2 372.3649} C_DIS
LIN {X 23.9412,Y 134.1678,Z 174,A 80.9227,B 7.8251,C 0.0948,E1 7.8542,E2 370.898} C_DIS
LIN {X 20.692,Y 134.7073,Z 174,A 82.324,B 7.8251,C 0.0939,E1 7.8504,E2 369.4952} C_DIS
LIN {X 16.976,Y 135.2278,Z 174,A 83.9653,B 7.8252,C 0.0922,E1 7.8458,E2 367.8467} C_DIS
LIN {X 13.1979,Y 135.6468,Z 174,A 85.5195,B 7.8252,C 0.0925,E1 7.8415,E2 366.2983} C_DIS
LIN {X 9.3476,Y 135.9676,Z 174,A 87.23,B 7.8252,C 0.0907,E1 7.8367,E2 364.5779} C_DIS
LIN {X 4.3336,Y 136.2195,Z 174,A 89.3244,B 7.8252,C 0.0907,E1 7.8309,E2 362.4864} C_DIS
LIN {X -0.2333,Y 136.2882,Z 174,A 91.1797,B 7.8252,C 0.0917,E1 7.8257,E2 360.6398} C_DIS
LIN {X -3.8885,Y 136.2319,Z 174,A 92.6848,B 7.8252,C 0.0924,E1 7.8215,E2 359.1394} C_DIS
LIN {X -7.8613,Y 136.0614,Z 174,A 94.4056,B 7.8252,C 0.0918,E1 7.8167,E2 357.4134} C_DIS
LIN {X -11.7757,Y 135.7779,Z 174,A 95.9829,B 7.8252,C 0.0934,E1 7.8123,E2 355.8459} C_DIS
LIN {X -15.7589,Y 135.3736,Z 174,A 97.7357,B 7.8252,C 0.0928,E1 7.8074,E2 354.0855} C_DIS
LIN {X -19.3514,Y 134.9063,Z 174,A 99.2159,B 7.8252,C 0.0941,E1 7.8034,E2 352.6113} C_DIS
LIN {X -23.0255,Y 134.3293,Z 174,A 100.8321,B 7.8252,C 0.094,E1 7.7989,E2 350.9896} C_DIS
LIN {X -26.9004,Y 133.6062,Z 174,A 102.5012,B 7.8252,C 0.0947,E1 7.7943,E2 349.32} C_DIS
LIN {X -30.5397,Y 132.8214,Z 174,A 104.0102,B 7.8252,C 0.0966,E1 7.7902,E2 347.8188} C_DIS
LIN {X -34.1401,Y 131.9432,Z 174,A 105.8364,B 7.8252,C 0.0934,E1 7.7852,E2 345.9609} C_DIS
LIN {X -38.6755,Y 130.6847,Z 174,A 107.569,B 7.8252,C 0.0989,E1 7.7806,E2 344.2598} C_DIS
LIN {X -41.6891,Y 129.7544,Z 174,A 108.9283,B 7.8252,C 0.0996,E1 7.777,E2 342.8973} C_DIS
LIN {X -45.1325,Y 128.598,Z 174,A 110.4552,B 7.8251,C 0.101,E1 7.773,E2 341.3714} C_DIS
LIN {X -50.2753,Y 126.6768,Z 174,A 112.7112,B 7.8251,C 0.1042,E1 7.7671,E2 339.1236} C_DIS
LIN {X -54.7304,Y 124.8165,Z 174,A 114.9594,B 7.8251,C 0.1031,E1 7.7613,E2 336.8502} C_DIS
LIN {X -61.5099,Y 121.6172,Z 174,A 117.8014,B 7.8249,C 0.1119,E1 7.7542,E2 334.0485} C_DIS
LIN {X -64.3341,Y 120.1491,Z 174,A 119.42,B 7.8249,C 0.1094,E1 7.7501,E2 332.3969} C_DIS
LIN {X -69.0657,Y 117.4929,Z 174,A 121.491,B 7.8249,C 0.1159,E1 7.7452,E2 330.3534} C_DIS
LIN {X -71.6886,Y 115.9117,Z 174,A 123.0371,B 7.8249,C 0.1139,E1 7.7414,E2 328.7768} C_DIS
LIN {X -75.2723,Y 113.6172,Z 174,A 124.8342,B 7.8249,C 0.1166,E1 7.7372,E2 326.9803} C_DIS
LIN {X -81.8891,Y 108.9443,Z 174,A 127.9691,B 7.8247,C 0.1264,E1 7.7302,E2 323.8816} C_DIS
LIN {X -84.9858,Y 106.5461,Z 174,A 129.9291,B 7.8247,C 0.1247,E1 7.7258,E2 321.8848} C_DIS
LIN {X -88.3865,Y 103.7424,Z 174,A 132.0297,B 7.8247,C 0.1246,E1 7.7212,E2 319.7555} C_DIS
LIN {X -90.8377,Y 101.6029,Z 174,A 132.9577,B 7.8247,C 0.1336,E1 7.7194,E2 318.8825} C_DIS
LIN {X -93.0996,Y 99.5348,Z 174,A 134.6134,B 7.8247,C 0.1308,E1 7.7159,E2 317.1831} C_DIS
LIN {X -97.017,Y 95.7209,Z 174,A 136.8139,B 7.8246,C 0.137,E1 7.7116,E2 314.9969} C_DIS
LIN {X -100.7744,Y 91.7562,Z 174,A 139.1609,B 7.8245,C 0.1411,E1 7.7071,E2 312.6458} C_DIS
LIN {X -103.9007,Y 88.2002,Z 174,A 141.1696,B 7.8245,C 0.1452,E1 7.7034,E2 310.6368} C_DIS
LIN {X -106.6946,Y 84.7992,Z 174,A 143.0671,B 7.8243,C 0.1487,E1 7.7001,E2 308.7353} C_DIS
LIN {X -109.3266,Y 81.3777,Z 174,A 144.9138,B 7.8243,C 0.1525,E1 7.697,E2 306.8864} C_DIS
LIN {X -111.9668,Y 77.7052,Z 174,A 146.8721,B 7.8242,C 0.1562,E1 7.6938,E2 304.9229} C_DIS
LIN {X -114.5251,Y 73.8836,Z 174,A 148.8417,B 7.8242,C 0.1603,E1 7.6908,E2 302.9509} C_DIS
LIN {X -117.0914,Y 69.7442,Z 174,A 151.4305,B 7.8242,C 0.1577,E1 7.687,E2 300.2971} C_DIS
LIN {X -119.5732,Y 65.3979,Z 174,A 153.1436,B 7.8239,C 0.1686,E1 7.6847,E2 298.6345} C_DIS
LIN {X -121.5718,Y 61.599,Z 174,A 154.741,B 7.8238,C 0.1762,E1 7.6827,E2 297.0643} C_DIS
LIN {X -122.9311,Y 58.8391,Z 174,A 156.1634,B 7.8238,C 0.1777,E1 7.681,E2 295.6273} C_DIS
LIN {X -124.6196,Y 55.1753,Z 174,A 157.8064,B 7.8236,C 0.183,E1 7.6791,E2 293.9925} C_DIS
LIN {X -125.8948,Y 52.1988,Z 174,A 159.3001,B 7.8236,C 0.1848,E1 7.6775,E2 292.4838} C_DIS
LIN {X -129.5889,Y 42.2072,Z 174,A 163.8202,B 7.8233,C 0.1965,E1 7.6732,E2 287.9633} C_DIS
LIN {X -130.9956,Y 37.6136,Z 174,A 165.8152,B 7.8231,C 0.2024,E1 7.6716,E2 285.9734} C_DIS
LIN {X -132.0297,Y 33.7991,Z 174,A 167.5793,B 7.8231,C 0.2056,E1 7.6703,E2 284.1981} C_DIS
LIN {X -132.9588,Y 29.9381,Z 174,A 169.2022,B 7.8229,C 0.211,E1 7.6693,E2 282.5826} C_DIS
LIN {X -133.7651,Y 26.1023,Z 174,A 170.9692,B 7.8229,C 0.214,E1 7.6683,E2 280.8024} C_DIS
LIN {X -134.4825,Y 22.1076,Z 174,A 172.6141,B 7.8227,C 0.2197,E1 7.6675,E2 279.1667} C_DIS
LIN {X -135.0285,Y 18.4968,Z 174,A 174.3507,B 7.8227,C 0.2213,E1 7.6669,E2 277.4067} C_DIS
LIN {X -135.5111,Y 14.5238,Z 174,A 175.9701,B 7.8225,C 0.227,E1 7.6663,E2 275.7966} C_DIS
LIN {X -135.8899,Y 10.4117,Z 174,A 177.7358,B 7.8223,C 0.2316,E1 7.6659,E2 274.0288} C_DIS
LIN {X -136.1157,Y 6.8381,Z 174,A 179.2378,B 7.8223,C 0.236,E1 7.6657,E2 272.5286} C_DIS
LIN {X -136.2635,Y 2.5689,Z 174,A -178.9155,B 7.8221,C 0.2405,E1 7.6656,E2 270.6771} C_DIS
LIN {X -136.2789,Y -1.642,Z 174,A -177.0729,B 7.8219,C 0.2446,E1 7.6656,E2 268.8271} C_DIS
LIN {X -136.1746,Y -5.5465,Z 174,A -175.4567,B 7.8218,C 0.2496,E1 7.6657,E2 267.2155} C_DIS
LIN {X -135.9416,Y -9.7037,Z 174,A -173.6308,B 7.8217,C 0.2536,E1 7.6661,E2 265.3817} C_DIS
LIN {X -135.6262,Y -13.4125,Z 174,A -172.0568,B 7.8215,C 0.258,E1 7.6665,E2 263.8079} C_DIS
LIN {X -135.1595,Y -17.4973,Z 174,A -170.3299,B 7.8214,C 0.2629,E1 7.667,E2 262.0825} C_DIS
LIN {X -134.6805,Y -20.8653,Z 174,A -168.8595,B 7.8212,C 0.2664,E1 7.6676,E2 260.6083} C_DIS
LIN {X -134.0087,Y -24.8281,Z 174,A -166.9916,B 7.8212,C 0.2687,E1 7.6686,E2 258.7194} C_DIS
LIN {X -133.1383,Y -29.129,Z 174,A -165.2232,B 7.8209,C 0.275,E1 7.6696,E2 256.962} C_DIS
LIN {X -132.1243,Y -33.4264,Z 174,A -162.114,B 7.8214,C 0.2624,E1 7.6719,E2 253.6958} C_DIS
LIN {X -129.8221,Y -41.4772,Z 174,A -160.106,B 7.8203,C 0.2935,E1 7.6734,E2 251.8814} C_DIS
LIN {X -128.478,Y -45.4769,Z 174,A -158.0149,B 7.8203,C 0.2938,E1 7.6753,E2 249.752} C_DIS
LIN {X -126.947,Y -49.5844,Z 174,A -156.0919,B 7.8201,C 0.2976,E1 7.6772,E2 247.8201} C_DIS
LIN {X -125.4927,Y -53.1618,Z 174,A -154.3092,B 7.8201,C 0.2996,E1 7.6791,E2 246.0184} C_DIS
LIN {X -123.3478,Y -57.9657,Z 174,A -152.2036,B 7.8198,C 0.3068,E1 7.6815,E2 243.9276} C_DIS
LIN {X -121.6863,Y -61.3741,Z 174,A -150.4894,B 7.8197,C 0.3092,E1 7.6837,E2 242.1992} C_DIS
LIN {X -119.8544,Y -64.8824,Z 174,A -148.6646,B 7.8196,C 0.311,E1 7.6861,E2 240.3551} C_DIS
LIN {X -118.1407,Y -67.9526,Z 174,A -147.3123,B 7.8194,C 0.3165,E1 7.688,E2 239.0195} C_DIS
LIN {X -115.9477,Y -71.6307,Z 174,A -145.4385,B 7.8192,C 0.3198,E1 7.6907,E2 237.1373} C_DIS
LIN {X -112.854,Y -76.4108,Z 174,A -143.0506,B 7.819,C 0.3255,E1 7.6943,E2 234.7513} C_DIS
Enddeposition()
END
